// TwinCAT 3 PLC project Untitled1
// ProgramVersion: 3.1.4026.24
// libraries:
//   RobustSolution, * (BATW)
//   Tc2_MC2, * (Beckhoff Automation GmbH)
//   Tc2_Standard, * (Beckhoff Automation GmbH)
//   Tc2_System, * (Beckhoff Automation GmbH)
//   TcUnit, * (www.tcunit.org)
// project tree:
//   GVLs/ GVL_IO.TcGVL (not stored), GVL_Module.TcGVL
//   / PlcTask.TcTTO, UnitTestTask.TcTTO
//   POUs/10_Chamber1/DUTs/Ctrl Status Interface/ ST_Chamber1_CtrlStatus.TcDUT, ST_Chamber1_ServiceCtrl.TcDUT, ST_Chamber1_ServiceParam.TcDUT, ST_Chamber1_ServiceStatus.TcDUT
//   POUs/10_Chamber1/DUTs/ E_Chamber1ErrorCode.TcDUT, E_Chamber1ServiceId.TcDUT
//   POUs/10_Chamber1/DUTs/External IO/ ST_Chamber1_Signal_In.TcDUT (not stored), ST_Chamber1_Signal_Out.TcDUT
//   POUs/10_Chamber1/DUTs/Service Param/PreparePositionService/ E_Chamber1PreparePositionStep.TcDUT (not stored), ST_Chamber1PreparePositionParam.TcDUT
//   POUs/10_Chamber1/DUTs/Service Param/ ST_Chamber1LiftPinAxisMoveAbsParam.TcDUT, ST_Chamber1LiftPinAxisMoveVelParam.TcDUT, ST_Chamber1SpinAxisJogParam.TcDUT, ST_Chamber1SpinAxisMoveAbsParam.TcDUT (not stored), ST_Chamber1SpinAxisMoveVelParam.TcDUT
//   POUs/10_Chamber1/ FB_Chamber1ModuleConfigurationAdapter.TcPOU (not stored), FB_Chamber1_Module.TcPOU
//   POUs/10_Chamber1/Services/ FB_Chamber1LiftPinAxisMoveAbsServices.TcPOU (not stored), FB_Chamber1LiftPinAxisMoveVelCCWServices.TcPOU (not stored), FB_Chamber1LiftPinAxisMoveVelCWServices.TcPOU (not stored), FB_Chamber1PreparePositionService.TcPOU (not stored), FB_Chamber1SpinAxisJogCWServices.TcPOU (not stored), FB_Chamber1SpinAxisMoveAbsServices.TcPOU (not stored), FB_Chamber1SpinAxisMoveVelCWServices.TcPOU (not stored), FB_Chamber1WaferReceiveService.TcPOU (not stored), FB_Chamber1WaferSendService.TcPOU
//   POUs/ FB_ConfigRoot.TcPOU, MAIN.TcPOU
//   Tests/DUTs/ E_FakeAxisOperation.TcDUT (not stored), ST_FakeAxisCall.TcDUT (not stored), ST_FakeAxisScriptStep.TcDUT (not stored)
//   Tests/Fakes/ FB_FakeAxis_BaseUnit.TcPOU (not stored)
//   Tests/ PRG_TEST.TcPOU
//   Tests/Suites/BaseUnit/ FB_FakeAxis_BaseUnitTests.TcPOU (not stored)
//   Tests/Suites/Modules/ FB_Chamber1_ModuleTests.TcPOU
//   Tests/Suites/Services/ FB_Chamber1MoveVelServiceTests.TcPOU, FB_Chamber1SpinAxisMoveAbsServiceTests.TcPOU
// real-time tasks:
//   TASK PlcTask: cycle T#10ms, priority 20, ADS port 350
//   TASK UnitTest Task: cycle T#10ms, priority 1, ADS port 351
// motion (NC):
//   TASK NC-Task 1 SAF: cycle T#2ms, priority 4, ADS port 501
//   TASK NC-Task 1 SVB: cycle T#10ms, priority 8, ADS port 511
//   AXIS Axis 1 (id 1)
//     OtherSettings: AllowMotionCmdToSlave=true
//     encoder EncType=1
//     drive DrvType=5
//       Analog: TorqueSetpointScale=10, ScaleFactorActTorque=0.1
//     controller CtrType=1
//       CtrPara: PriorControlFactor=1
//         Observer: BandWidth=20
//   AXIS Axis 2 (id 2)
//     OtherSettings: AllowMotionCmdToSlave=true
//     encoder EncType=1
//     drive DrvType=5
//       Analog: TorqueSetpointScale=10, ScaleFactorActTorque=0.1
//     controller CtrType=1
//       CtrPara: PriorControlFactor=1
//         Observer: BandWidth=20
// variable links:
//   Untitled1/Untitled1 Instance <-> NC-Task 1 SAF/Axes/Axis 1
//     PlcTask Inputs/GVL_IO.NC_Axis1._Axis.NcToPlc <-> Outputs/ToPlc
//     PlcTask Outputs/GVL_IO.NC_Axis1._Axis.PlcToNc <-> Inputs/FromPlc
//   Untitled1/Untitled1 Instance <-> NC-Task 1 SAF/Axes/Axis 2
//     PlcTask Inputs/GVL_IO.NC_Axis2._Axis.NcToPlc <-> Outputs/ToPlc
//     PlcTask Outputs/GVL_IO.NC_Axis2._Axis.PlcToNc <-> Inputs/FromPlc

CONFIGURATION Untitled1
    RESOURCE PLC ON TwinCAT3
        TASK PlcTask(INTERVAL := T#10ms, PRIORITY := 20);
        TASK UnitTestTask(INTERVAL := T#10ms, PRIORITY := 1);
        PROGRAM MAIN WITH PlcTask : MAIN;
        PROGRAM PRG_TEST WITH UnitTestTask : PRG_TEST;
    END_RESOURCE
END_CONFIGURATION

// ---- POUs/10_Chamber1/DUTs/Ctrl Status Interface/ST_Chamber1_CtrlStatus.TcDUT
TYPE ST_Chamber1_CtrlStatus EXTENDS ST_Module_CtrlStatus_Base :
STRUCT
	ServiceCtrl : ST_Chamber1_ServiceCtrl;
	ServiceParam : ST_Chamber1_ServiceParam;
	ServiceStatus : ST_Chamber1_ServiceStatus;
END_STRUCT
END_TYPE

// ---- POUs/10_Chamber1/DUTs/Ctrl Status Interface/ST_Chamber1_ServiceCtrl.TcDUT
TYPE ST_Chamber1_ServiceCtrl :
STRUCT
	SpinAxisJogCW : ST_ServiceCtrl;
	SpinAxisMoveAbs : ST_ServiceCtrl;
	SpinAxisMoveVelCW	: ST_ServiceCtrl;
	LiftPinAxisMoveVelCW : ST_ServiceCtrl;
	LiftPinAxisMoveVelCCW : ST_ServiceCtrl;
	LiftPinAxisMoveAbs : ST_ServiceCtrl;
	
	WaferSend : ST_ServiceCtrl;
	WaferReceive : ST_ServiceCtrl;
	PreparePosition : ST_ServiceCtrl;
END_STRUCT
END_TYPE

// ---- POUs/10_Chamber1/DUTs/Ctrl Status Interface/ST_Chamber1_ServiceParam.TcDUT
TYPE ST_Chamber1_ServiceParam :
STRUCT
	SpinAxisJogCW : ST_Chamber1SpinAxisJogParam;
	SpinAxisMoveAbs : ST_Chamber1SpinAxisMoveAbsParam;
	SpinAxisMoveVelCW : ST_Chamber1SpinAxisMoveVelParam;
	LiftPinAxisMoveVelCW : ST_Chamber1LiftPinAxisMoveVelParam;
	LiftPinAxisMoveVelCCW : ST_Chamber1LiftPinAxisMoveVelParam;
	LiftPinAxisMoveAbs : ST_Chamber1LiftPinAxisMoveAbsParam;
	WaferReceive : ST_WaferTransferParam;
	WaferSend : ST_WaferTransferParam;
	PreparePosition : ST_Chamber1PreparePositionParam;
END_STRUCT
END_TYPE

// ---- POUs/10_Chamber1/DUTs/Ctrl Status Interface/ST_Chamber1_ServiceStatus.TcDUT
TYPE ST_Chamber1_ServiceStatus :
STRUCT
	SpinAxisJogCW : ST_ServiceStatus;
	SpinAxisMoveAbs : ST_ServiceStatus;
	SpinAxisMoveVelCW : ST_ServiceStatus;
	LiftPinAxisMoveVelCW : ST_ServiceStatus;
	LiftPinAxisMoveVelCCW : ST_ServiceStatus;
	LiftPinAxisMoveAbs : ST_ServiceStatus;
	WaferSend : ST_ServiceStatus;
	WaferReceive : ST_ServiceStatus;
	PreparePosition : ST_ServiceStatus;
END_STRUCT
END_TYPE

// ---- POUs/10_Chamber1/DUTs/E_Chamber1ErrorCode.TcDUT
{attribute 'qualified_only'}
{attribute 'to_string'}
TYPE E_Chamber1ErrorCode :
(
	None := 0,
	Axis_Not_Servo_On_During_Starting := 1,
	Axis_Is_Busy_During_Starting := 2,
	Invalid_Param := 3,
	Axis_Command_Error_During_Execute := 4,
	Error_While_Stop_Axis := 5,
	// The BaseUnit was already owned by another Service.
	Resource_Acquire_Failed_During_Starting := 6,
	// The asynchronous Reset used while aborting failed.
	Error_While_Reset_Axis := 7
)UDINT;
END_TYPE

// ---- POUs/10_Chamber1/DUTs/E_Chamber1ServiceId.TcDUT
{attribute 'qualified_only'}
{attribute 'to_string'}
TYPE E_Chamber1ServiceId :
(
	// Each value identifies one Service instance within the Chamber1 Module.
	None := 0,
	SpinAxisJogCW := 1,
	SpinAxisMoveAbs := 2,
	SpinAxisMoveVelCW := 3,
	LiftPinAxisMoveVelCW := 4,
	LiftPinAxisMoveVelCCW := 5,
	LiftPinAxisMoveAbs := 6,
	WaferSend := 8,
	WaferReceive := 9,
	PreparePosition := 10
) UDINT;
END_TYPE

// ---- POUs/10_Chamber1/DUTs/External IO/ST_Chamber1_Signal_Out.TcDUT
TYPE ST_Chamber1_Signal_Out :
STRUCT
	bVaccumOn : BOOL;

	bDOs : ARRAY[1..16] OF BOOL;
	rAOs : ARRAY[1..16] OF REAL;
END_STRUCT
END_TYPE

// ---- POUs/10_Chamber1/DUTs/Service Param/PreparePositionService/ST_Chamber1PreparePositionParam.TcDUT
TYPE ST_Chamber1PreparePositionParam :
STRUCT
	LiftReady : ST_Chamber1LiftPinAxisMoveAbsParam;
	SpinAlign : ST_Chamber1SpinAxisMoveAbsParam;
	LiftWork : ST_Chamber1LiftPinAxisMoveAbsParam;
END_STRUCT
END_TYPE

// ---- POUs/10_Chamber1/DUTs/Service Param/ST_Chamber1LiftPinAxisMoveAbsParam.TcDUT
TYPE ST_Chamber1LiftPinAxisMoveAbsParam :
STRUCT
	Position : LREAL;
	Velocity : LREAL;
	Acceleration : LREAL;
	Deceleration : LREAL;
END_STRUCT
END_TYPE

// ---- POUs/10_Chamber1/DUTs/Service Param/ST_Chamber1LiftPinAxisMoveVelParam.TcDUT
TYPE ST_Chamber1LiftPinAxisMoveVelParam :
STRUCT
	Velocity : LREAL;
	Acceleration : LREAL;
	Deceleration : LREAL;
END_STRUCT
END_TYPE

// ---- POUs/10_Chamber1/DUTs/Service Param/ST_Chamber1SpinAxisJogParam.TcDUT
TYPE ST_Chamber1SpinAxisJogParam :
STRUCT
	Position : LREAL;
	Velocity : LREAL;
	Acceleration : LREAL;
	Deceleration : LREAL;
END_STRUCT
END_TYPE

// ---- POUs/10_Chamber1/DUTs/Service Param/ST_Chamber1SpinAxisMoveVelParam.TcDUT
TYPE ST_Chamber1SpinAxisMoveVelParam :
STRUCT
	Velocity : LREAL;
	Acceleration : LREAL;
	Deceleration : LREAL;
END_STRUCT
END_TYPE

// ---- GVLs/GVL_Module.TcGVL
{attribute 'qualified_only'}
VAR_GLOBAL
	Chamber1 : ARRAY[1..Param_Config.MaxModulePerType] OF FB_Chamber1_Module;
	Chamber1_Runtime : ARRAY[1..Param_Config.MaxModulePerType] OF ST_ModuleRuntimeConfig;
	Chamber1_Control : ARRAY[1..Param_Config.MaxModulePerType] OF ST_Chamber1_CtrlStatus;
	Chamber1_SpinAxis : ARRAY[1..Param_Config.MaxModulePerType] OF I_Axis_BaseUnit;
	Chamber1_LiftPinAxis : ARRAY[1..Param_Config.MaxModulePerType] OF I_Axis_BaseUnit;
END_VAR

// ---- POUs/MAIN.TcPOU
PROGRAM MAIN
VAR
	ConfigRoot : FB_ConfigRoot;
END_VAR

ConfigRoot.Run();

END_PROGRAM

// ---- POUs/FB_ConfigRoot.TcPOU
FUNCTION_BLOCK FB_ConfigRoot EXTENDS FB_ApplicationConfigRoot
VAR
	_Chamber1ModuleConfigurationAdapter : FB_Chamber1ModuleConfigurationAdapter;
END_VAR

METHOD PROTECTED H_RegisterBaseUnits
M_RegisterBaseUnit(BaseUnit := GVL_IO.NC_Axis1);
M_RegisterBaseUnit(BaseUnit := GVL_IO.NC_Axis2);
END_METHOD

METHOD PROTECTED H_RegisterIo
VAR
	nChannel : DINT;
END_VAR
FOR nChannel := LOWER_BOUND(GVL_IO.Term4_EL1889.Chl, 1)
	TO UPPER_BOUND(GVL_IO.Term4_EL1889.Chl, 1) DO
	IF NOT M_RegisterIoNode(
		Variable := GVL_IO.Term4_EL1889.Chl[nChannel],
		Access := E_VariableAccess.ReadOnly) THEN
		RETURN;
	END_IF
END_FOR

FOR nChannel := LOWER_BOUND(GVL_IO.Term2_EL3602.Chl, 1)
	TO UPPER_BOUND(GVL_IO.Term2_EL3602.Chl, 1) DO
	IF NOT M_RegisterIoNode(
		Variable := GVL_IO.Term2_EL3602.Chl[nChannel],
		Access := E_VariableAccess.ReadOnly) THEN
		RETURN;
	END_IF
END_FOR

FOR nChannel := LOWER_BOUND(GVL_IO.Term3_EL2809.Chl, 1)
	TO UPPER_BOUND(GVL_IO.Term3_EL2809.Chl, 1) DO
	IF NOT M_RegisterIoNode(
		Variable := GVL_IO.Term3_EL2809.Chl[nChannel],
		Access := E_VariableAccess.WriteOnly) THEN
		RETURN;
	END_IF
END_FOR
END_METHOD

METHOD PROTECTED H_RegisterModuleTypes
M_RegisterModuleType(
	ModuleTypeName := 'Chamber1',
	Adapter := _Chamber1ModuleConfigurationAdapter);
END_METHOD

METHOD PROTECTED H_RunModules
VAR_INPUT
	VariableNodeReader : I_VariableNodeReader;
END_VAR
VAR_IN_OUT CONSTANT
	SystemContext : ST_SystemContext;
END_VAR
VAR
	nModule : UINT;
END_VAR
FOR nModule := 1 TO Param_Config.MaxModulePerType DO
	IF GVL_Module.Chamber1_Runtime[nModule].Enabled
		AND GVL_Module.Chamber1_Runtime[nModule].Valid THEN
		GVL_Module.Chamber1[nModule](
			HeartbeatIndex := GVL_Module.Chamber1_Control[nModule].HeartbeatIndex,
			ModuleCtrl := GVL_Module.Chamber1_Control[nModule].ModuleCtrl,
			ServiceCtrl := GVL_Module.Chamber1_Control[nModule].ServiceCtrl,
			ServiceParam := GVL_Module.Chamber1_Control[nModule].ServiceParam,
			SystemContext := SystemContext,
			RuntimeConfig := GVL_Module.Chamber1_Runtime[nModule],
			VariableNodeReader := VariableNodeReader,
			SpinAxis_BaseUnit := GVL_Module.Chamber1_SpinAxis[nModule],
			LiftPinAxis_BaseUnit := GVL_Module.Chamber1_LiftPinAxis[nModule],
			ModuleStatus => GVL_Module.Chamber1_Control[nModule].ModuleStatus,
			ServiceStatus => GVL_Module.Chamber1_Control[nModule].ServiceStatus,
			ModuleAlarmList => GVL_Module.Chamber1_Control[nModule].ModuleAlarmList,
			ModuleDataList => GVL_Module.Chamber1_Control[nModule].ModuleDataList,
			ModuleVariableList => GVL_Module.Chamber1_Control[nModule].ModuleVariableList);
	END_IF
END_FOR
END_METHOD

END_FUNCTION_BLOCK

// ---- Tests/PRG_TEST.TcPOU
PROGRAM PRG_TEST
VAR
	FakeAxisContractTests : FB_FakeAxis_BaseUnitTests;
	
	MoveAbsServiceTests : FB_Chamber1SpinAxisMoveAbsServiceTests;
	MoveVelServiceTests : FB_Chamber1MoveVelServiceTests;
	
	Chamber1ModuleTests : FB_Chamber1_ModuleTests;
END_VAR

TcUnit.RUN();

END_PROGRAM

// ---- Tests/Suites/Services/FB_Chamber1SpinAxisMoveAbsServiceTests.TcPOU
FUNCTION_BLOCK FB_Chamber1SpinAxisMoveAbsServiceTests EXTENDS TcUnit.FB_TestSuite

SuccessfulMoveAbsCompletesAndReleasesAxis();
MoveAbsErrorStopsSafelyAndRecordsError();
InvalidParamStopsStartingWithoutAcquiringAxis();
ResourceAcquireFailureStopsStartingWithoutDisturbingOwner();

METHOD InvalidParamStopsStartingWithoutAcquiringAxis
VAR_INST
	FakeAxis : FB_FakeAxis_BaseUnit;
	Axis : I_Axis_BaseUnit;
	Service : FB_Chamber1SpinAxisMoveAbsServices;
	Ctrl : ST_ServiceCtrl;
	Param : ST_Chamber1SpinAxisMoveAbsParam;
	Context : ST_ServiceContext;
	nPhase : UINT;
END_VAR
TEST('InvalidParamStopsStartingWithoutAcquiringAxis');

CASE nPhase OF
	0:
		// Set invalid param
		FakeAxis.M_ResetScenario();
		Axis := FakeAxis;
		Param.Position := 50;
		Param.Velocity := 0;
		Param.Acceleration := 20;
		Param.Deceleration := 30;
		Context.ModuleId := 1;
		Context.UtcDateTime := '20260813123456007';

		// Cyclic update
		Service(Ctrl := Ctrl, Param := Param, Context := Context, Axis_BaseUnit := Axis, ServiceId := 23);
		FakeAxis.M_CyclicUpdate();

		// Check service run into certain state
		AssertTrue(Condition := Service.PackMLOut.eStateCurrent = E_PackMLState.Aborted, Message := 'Initial scan must reach Aborted.');
		nPhase := 1;

	1:
		// Set PackML cmd: Clear
		Ctrl.PackMLIn.eCommand := E_PackMLCommand.Clear;
		Ctrl.PackMLIn.bCommandChangeRequest := TRUE;

		// Cyclic update
		Service(Ctrl := Ctrl, Param := Param, Context := Context, Axis_BaseUnit := Axis, ServiceId := 23);
		FakeAxis.M_CyclicUpdate();

		// Check service run into certain state
		AssertTrue(Condition := Service.PackMLOut.eStateCurrent = E_PackMLState.Stopped, Message := 'Clear must reach Stopped.');

		// Reset request flag
		Ctrl.PackMLIn.bCommandChangeRequest := FALSE;
		Service(Ctrl := Ctrl, Param := Param, Context := Context, Axis_BaseUnit := Axis, ServiceId := 23);
		FakeAxis.M_CyclicUpdate();

		// Set PackML cmd: Reset
		Ctrl.PackMLIn.eCommand := E_PackMLCommand.Reset;
		Ctrl.PackMLIn.bCommandChangeRequest := TRUE;

		// Cyclic update
		Service(Ctrl := Ctrl, Param := Param, Context := Context, Axis_BaseUnit := Axis, ServiceId := 23);
		FakeAxis.M_CyclicUpdate();

		// Check service run into certain state
		AssertTrue(Condition := Service.PackMLOut.eStateCurrent = E_PackMLState.Idle, Message := 'Reset must reach Idle.');
		nPhase := 2;

	2:
		// Reset request flag
		Ctrl.PackMLIn.bCommandChangeRequest := FALSE;
		Service(Ctrl := Ctrl, Param := Param, Context := Context, Axis_BaseUnit := Axis, ServiceId := 23);
		FakeAxis.M_CyclicUpdate();

		// Set PackML cmd: Start
		Ctrl.PackMLIn.eCommand := E_PackMLCommand.Start;
		Ctrl.PackMLIn.bCommandChangeRequest := TRUE;

		// Cyclic update
		Service(Ctrl := Ctrl, Param := Param, Context := Context, Axis_BaseUnit := Axis, ServiceId := 23);
		FakeAxis.M_CyclicUpdate();

		// Check service remains in Starting until queued Stop is processed
		AssertTrue(Condition := Service.PackMLOut.eStateCurrent = E_PackMLState.Starting, Message := 'Invalid Param must remain in Starting until queued Stop is processed.');

		// Check certain alarm emerged
		AssertTrue(Condition := Service.Status.ErrorList[1].MainErrorId = E_Chamber1ErrorCode.Invalid_Param, Message := 'Invalid Velocity must record Invalid_Param.');
		AssertTrue(Condition := Service.Status.ErrorList[1].SourceErrorId = 0, Message := 'Invalid Param must use SourceErrorId zero.');
		AssertTrue(Condition := Service.Status.ErrorList[1].Message = 'Velocity must be greater than zero.', Message := 'Invalid Velocity must have a specific message.');

		// Check service did not acquire or call the Axis
		AssertFalse(Condition := Axis.M_IsResourceOwner(OwnerId := 23), Message := 'Invalid Param must not acquire Axis ownership.');
		AssertTrue(Condition := FakeAxis.HistoryCount = 0, Message := 'Invalid Param must not issue an Axis command.');
		nPhase := 3;

	3:
		// Reset request flag & process queued Stop
		Ctrl.PackMLIn.bCommandChangeRequest := FALSE;
		Service(Ctrl := Ctrl, Param := Param, Context := Context, Axis_BaseUnit := Axis, ServiceId := 23);
		FakeAxis.M_CyclicUpdate();

		// Check service safely returns to Stopped
		AssertTrue(Condition := Service.PackMLOut.eStateCurrent = E_PackMLState.Stopped, Message := 'Queued Stop must return invalid Starting to Stopped.');

		// Check no duplicate alarm or Axis side effect emerged
		AssertTrue(Condition := Service.Status.ErrorList[1].MainErrorId = E_Chamber1ErrorCode.Invalid_Param, Message := 'Invalid Param must remain recorded after stopping.');
		AssertTrue(Condition := Service.Status.ErrorList[2].MainErrorId = 0, Message := 'Invalid Param must only be recorded once.');
		AssertFalse(Condition := Axis.M_IsResourceOwner(OwnerId := 23), Message := 'Stopped Service must not own the Axis.');
		AssertTrue(Condition := FakeAxis.HistoryCount = 0, Message := 'Stopping without ownership must not issue an Axis command.');
		nPhase := 0;

		TEST_FINISHED();
END_CASE
END_METHOD

METHOD MoveAbsErrorStopsSafelyAndRecordsError
VAR_INST
	FakeAxis : FB_FakeAxis_BaseUnit;
	Axis : I_Axis_BaseUnit;
	Service : FB_Chamber1SpinAxisMoveAbsServices;
	Ctrl : ST_ServiceCtrl;
	Param : ST_Chamber1SpinAxisMoveAbsParam;
	Context : ST_ServiceContext;
	MoveWithdrawalCall : ST_FakeAxisCall;
	StopCall : ST_FakeAxisCall;
	nHistoryBeforeStopping : UINT;
	nPhase : UINT;
END_VAR
TEST('MoveAbsErrorStopsSafelyAndRecordsError');

CASE nPhase OF
	0:
		// Set param
		FakeAxis.M_ResetScenario();
		Axis := FakeAxis;
		Param.Position := 50;
		Param.Velocity := 10;
		Param.Acceleration := 20;
		Param.Deceleration := 30;
		Context.ModuleId := 1;
		Context.UtcDateTime := '20260813123456007';
		
		// Set script: move abs. failed and then stop success
		AssertTrue(
			Condition := FakeAxis.M_QueueResult(
				Operation := E_FakeAxisOperation.MoveAbs,
				AfterActiveCycles := 1,
				Done := FALSE,
				InVelocity := FALSE,
				Error := TRUE,
				ErrorId := 16#1234),
			Message := 'MoveAbs Error script must be accepted.');
		AssertTrue(
			Condition := FakeAxis.M_QueueResult(
				Operation := E_FakeAxisOperation.Stop,
				AfterActiveCycles := 2,
				Done := TRUE,
				InVelocity := FALSE,
				Error := FALSE,
				ErrorId := 0),
			Message := 'Stop Done script must be accepted.');
		
		// Cyclic update
		Service(Ctrl := Ctrl, Param := Param, Context := Context, Axis_BaseUnit := Axis, ServiceId := 22);
		FakeAxis.M_CyclicUpdate();
		nPhase := 1;

	1:
		// Set PackML cmd: Clear
		Ctrl.PackMLIn.eCommand := E_PackMLCommand.Clear;
		Ctrl.PackMLIn.bCommandChangeRequest := TRUE;
		Service(Ctrl := Ctrl, Param := Param, Context := Context, Axis_BaseUnit := Axis, ServiceId := 22);
		FakeAxis.M_CyclicUpdate();

		// Reset request flag
		Ctrl.PackMLIn.bCommandChangeRequest := FALSE;
		Service(Ctrl := Ctrl, Param := Param, Context := Context, Axis_BaseUnit := Axis, ServiceId := 22);
		FakeAxis.M_CyclicUpdate();

		// Set PackML cmd: Reset
		Ctrl.PackMLIn.eCommand := E_PackMLCommand.Reset;
		Ctrl.PackMLIn.bCommandChangeRequest := TRUE;
		Service(Ctrl := Ctrl, Param := Param, Context := Context, Axis_BaseUnit := Axis, ServiceId := 22);
		FakeAxis.M_CyclicUpdate();
		nPhase := 2;

	2:
		// Reset request flag
		Ctrl.PackMLIn.bCommandChangeRequest := FALSE;
		Service(Ctrl := Ctrl, Param := Param, Context := Context, Axis_BaseUnit := Axis, ServiceId := 22);
		FakeAxis.M_CyclicUpdate();

		// Set PackML cmd: Start
		Ctrl.PackMLIn.eCommand := E_PackMLCommand.Start;
		Ctrl.PackMLIn.bCommandChangeRequest := TRUE;
		Service(Ctrl := Ctrl, Param := Param, Context := Context, Axis_BaseUnit := Axis, ServiceId := 22);
		FakeAxis.M_CyclicUpdate();
		AssertTrue(Condition := Service.PackMLOut.eStateCurrent = E_PackMLState.Execute, Message := 'Start must reach Execute.');
		nPhase := 3;

	3:
		// Reset request flag & 1st call of move abs. !!!
		Ctrl.PackMLIn.bCommandChangeRequest := FALSE;
		Service(Ctrl := Ctrl, Param := Param, Context := Context, Axis_BaseUnit := Axis, ServiceId := 22);
		FakeAxis.M_CyclicUpdate();
		AssertTrue(Condition := Service.PackMLOut.eStateCurrent = E_PackMLState.Execute, Message := 'MoveAbs Error is reported after the scripted active scan.');
		nPhase := 4;

	4:
		// 2nd call of move abs., error should happened
		Service(Ctrl := Ctrl, Param := Param, Context := Context, Axis_BaseUnit := Axis, ServiceId := 22);
		FakeAxis.M_CyclicUpdate();
		
		// Check service run into certain state
		AssertTrue(Condition := Service.PackMLOut.eStateCurrent = E_PackMLState.Execute, Message := 'MoveAbs Error must queue Stop for the next scan.');
		
		// Check certain alarm emerged
		AssertTrue(Condition := Service.Status.ErrorList[1].MainErrorId = E_Chamber1ErrorCode.Axis_Command_Error_During_Execute, Message := 'MoveAbs Error must be recorded.');
		AssertTrue(Condition := Service.Status.ErrorList[1].SourceErrorId = 16#1234, Message := 'MoveAbs Error must preserve the Axis source error ID.');
		AssertTrue(Condition := Service.Status.ErrorList[2].MainErrorId = 0, Message := 'MoveAbs Error must only be recorded once.');
		AssertTrue(Condition := Axis.M_IsResourceOwner(OwnerId := 22), Message := 'Queued Stop must retain ownership.');
		nPhase := 5;

	5:
		nHistoryBeforeStopping := FakeAxis.HistoryCount;
		
		// Cyclic update
		Service(Ctrl := Ctrl, Param := Param, Context := Context, Axis_BaseUnit := Axis, ServiceId := 22);
		FakeAxis.M_CyclicUpdate();
		
		// Check service run into certain state
		AssertTrue(Condition := Service.PackMLOut.eStateCurrent = E_PackMLState.Stopping, Message := 'Queued Stop must enter Stopping on the next scan.');
		
		// Check withdrawal move abs. cmd
		AssertTrue(Condition := FakeAxis.M_GetCall(Index := nHistoryBeforeStopping + 1, CallRecord => MoveWithdrawalCall), Message := 'Stopping must record MoveAbs withdrawal.');
		AssertTrue(Condition := MoveWithdrawalCall.Operation = E_FakeAxisOperation.MoveAbs, Message := 'Stopping must withdraw MoveAbs before Stop.');
		AssertTrue(Condition := MoveWithdrawalCall.Accepted, Message := 'MoveAbs withdrawal must be accepted.');
		AssertFalse(Condition := MoveWithdrawalCall.Execute, Message := 'Stopping must set MoveAbs Execute to FALSE.');
		
		// Check stop cmd has been called
		AssertTrue(Condition := FakeAxis.M_GetCall(Index := nHistoryBeforeStopping + 2, CallRecord => StopCall), Message := 'Stopping must record Stop after MoveAbs withdrawal.');
		AssertTrue(Condition := StopCall.Operation = E_FakeAxisOperation.Stop, Message := 'Stopping must issue Stop after MoveAbs withdrawal.');
		AssertTrue(Condition := StopCall.Accepted, Message := 'Stop must be accepted by the owned Axis.');
		AssertTrue(Condition := StopCall.Execute, Message := 'Stop Execute must be TRUE while pending.');
		AssertTrue(Condition := StopCall.Deceleration = Param.Deceleration, Message := 'Stop must preserve Deceleration.');
		AssertTrue(Condition := Axis.M_IsResourceOwner(OwnerId := 22), Message := 'Pending Stop must retain ownership.');
		nPhase := 6;

	6:
		// Cyclic update
		Service(Ctrl := Ctrl, Param := Param, Context := Context, Axis_BaseUnit := Axis, ServiceId := 22);
		FakeAxis.M_CyclicUpdate();
		
		// Stop cmd not finished yet according to script
		AssertTrue(Condition := Service.PackMLOut.eStateCurrent = E_PackMLState.Stopping, Message := 'Stop must remain Stopping until Done feedback is observed.');
		AssertTrue(Condition := Axis.M_IsResourceOwner(OwnerId := 22), Message := 'Stop pending scan must retain ownership.');
		nPhase := 7;

	7:
		// Cyclic update
		Service(Ctrl := Ctrl, Param := Param, Context := Context, Axis_BaseUnit := Axis, ServiceId := 22);
		FakeAxis.M_CyclicUpdate();
		
		// Check service run into certain state
		AssertTrue(Condition := Service.PackMLOut.eStateCurrent = E_PackMLState.Stopped, Message := 'Stop Done must reach Stopped.');
		
		// Check resource has been released
		AssertFalse(Condition := Axis.M_IsResourceOwner(OwnerId := 22), Message := 'Stop Done must release Axis ownership.');
		
		// Check alarm still exist
		AssertTrue(Condition := Service.Status.ErrorList[1].MainErrorId = E_Chamber1ErrorCode.Axis_Command_Error_During_Execute, Message := 'MoveAbs Error must remain recorded after stopping.');
		AssertTrue(Condition := Service.Status.ErrorList[1].SourceErrorId = 16#1234, Message := 'Recorded MoveAbs source error ID must remain unchanged.');
		AssertTrue(Condition := Service.Status.ErrorList[2].MainErrorId = 0, Message := 'Repeated scans must not duplicate the MoveAbs Error.');
		
		// Check withdrawal stop cmd
		AssertTrue(Condition := FakeAxis.M_GetCall(Index := FakeAxis.HistoryCount, CallRecord => StopCall), Message := 'Stop falling edge must be recorded.');
		AssertTrue(Condition := StopCall.Operation = E_FakeAxisOperation.Stop, Message := 'Final cleanup call must be Stop.');
		AssertTrue(Condition := StopCall.Accepted, Message := 'Stop falling edge must occur before ownership is released.');
		AssertFalse(Condition := StopCall.Execute, Message := 'Stop Done must set Stop Execute to FALSE.');
		AssertFalse(Condition := FakeAxis.HistoryOverflowed, Message := 'Fake Axis call history must not overflow.');
		nPhase := 0;
		
		TEST_FINISHED();
END_CASE
END_METHOD

METHOD ResourceAcquireFailureStopsStartingWithoutDisturbingOwner
VAR_INST
	FakeAxis : FB_FakeAxis_BaseUnit;
	Axis : I_Axis_BaseUnit;
	Service : FB_Chamber1SpinAxisMoveAbsServices;
	Ctrl : ST_ServiceCtrl;
	Param : ST_Chamber1SpinAxisMoveAbsParam;
	Context : ST_ServiceContext;
	nPhase : UINT;
END_VAR
TEST('ResourceAcquireFailureStopsStartingWithoutDisturbingOwner');

CASE nPhase OF
	0:
		// Set valid param
		FakeAxis.M_ResetScenario();
		Axis := FakeAxis;
		Param.Position := 50;
		Param.Velocity := 10;
		Param.Acceleration := 20;
		Param.Deceleration := 30;
		Context.ModuleId := 1;
		Context.UtcDateTime := '20260813123456007';

		// Cyclic update
		Service(Ctrl := Ctrl, Param := Param, Context := Context, Axis_BaseUnit := Axis, ServiceId := 24);
		FakeAxis.M_CyclicUpdate();

		// Check service run into certain state
		AssertTrue(Condition := Service.PackMLOut.eStateCurrent = E_PackMLState.Aborted, Message := 'Initial scan must reach Aborted.');
		nPhase := 1;

	1:
		// Set PackML cmd: Clear
		Ctrl.PackMLIn.eCommand := E_PackMLCommand.Clear;
		Ctrl.PackMLIn.bCommandChangeRequest := TRUE;

		// Cyclic update
		Service(Ctrl := Ctrl, Param := Param, Context := Context, Axis_BaseUnit := Axis, ServiceId := 24);
		FakeAxis.M_CyclicUpdate();

		// Check service run into certain state
		AssertTrue(Condition := Service.PackMLOut.eStateCurrent = E_PackMLState.Stopped, Message := 'Clear must reach Stopped.');

		// Reset request flag
		Ctrl.PackMLIn.bCommandChangeRequest := FALSE;
		Service(Ctrl := Ctrl, Param := Param, Context := Context, Axis_BaseUnit := Axis, ServiceId := 24);
		FakeAxis.M_CyclicUpdate();

		// Set PackML cmd: Reset
		Ctrl.PackMLIn.eCommand := E_PackMLCommand.Reset;
		Ctrl.PackMLIn.bCommandChangeRequest := TRUE;

		// Cyclic update
		Service(Ctrl := Ctrl, Param := Param, Context := Context, Axis_BaseUnit := Axis, ServiceId := 24);
		FakeAxis.M_CyclicUpdate();

		// Check service run into certain state
		AssertTrue(Condition := Service.PackMLOut.eStateCurrent = E_PackMLState.Idle, Message := 'Reset must reach Idle.');
		nPhase := 2;

	2:
		// Reset request flag
		Ctrl.PackMLIn.bCommandChangeRequest := FALSE;
		Service(Ctrl := Ctrl, Param := Param, Context := Context, Axis_BaseUnit := Axis, ServiceId := 24);
		FakeAxis.M_CyclicUpdate();

		// Reserve the Axis with another owner
		AssertTrue(Condition := Axis.M_AcquireResource(OwnerId := 99), Message := 'Another owner must reserve the Axis.');

		// Set PackML cmd: Start
		Ctrl.PackMLIn.eCommand := E_PackMLCommand.Start;
		Ctrl.PackMLIn.bCommandChangeRequest := TRUE;

		// Cyclic update
		Service(Ctrl := Ctrl, Param := Param, Context := Context, Axis_BaseUnit := Axis, ServiceId := 24);
		FakeAxis.M_CyclicUpdate();

		// Check service remains in Starting until queued Stop is processed
		AssertTrue(Condition := Service.PackMLOut.eStateCurrent = E_PackMLState.Starting, Message := 'Resource acquire failure must remain in Starting until queued Stop is processed.');

		// Check certain alarm emerged
		AssertTrue(Condition := Service.Status.ErrorList[1].MainErrorId = E_Chamber1ErrorCode.Resource_Acquire_Failed_During_Starting, Message := 'Resource contention must be recorded.');
		AssertTrue(Condition := Service.Status.ErrorList[1].SourceErrorId = 0, Message := 'Resource contention must use SourceErrorId zero.');

		// Check existing ownership was not disturbed
		AssertFalse(Condition := Axis.M_IsResourceOwner(OwnerId := 24), Message := 'Service must not acquire the reserved Axis.');
		AssertTrue(Condition := Axis.M_IsResourceOwner(OwnerId := 99), Message := 'Existing Axis owner must remain unchanged.');
		AssertTrue(Condition := FakeAxis.HistoryCount = 0, Message := 'Acquire failure must not issue an Axis command.');
		nPhase := 3;

	3:
		// Reset request flag & process queued Stop
		Ctrl.PackMLIn.bCommandChangeRequest := FALSE;
		Service(Ctrl := Ctrl, Param := Param, Context := Context, Axis_BaseUnit := Axis, ServiceId := 24);
		FakeAxis.M_CyclicUpdate();

		// Check service safely returns to Stopped
		AssertTrue(Condition := Service.PackMLOut.eStateCurrent = E_PackMLState.Stopped, Message := 'Queued Stop must return resource failure to Stopped.');

		// Check existing ownership and alarm remain unchanged
		AssertFalse(Condition := Axis.M_IsResourceOwner(OwnerId := 24), Message := 'Stopped Service must not own the Axis.');
		AssertTrue(Condition := Axis.M_IsResourceOwner(OwnerId := 99), Message := 'Stopping must not release another owner resource.');
		AssertTrue(Condition := Service.Status.ErrorList[1].MainErrorId = E_Chamber1ErrorCode.Resource_Acquire_Failed_During_Starting, Message := 'Resource contention must remain recorded after stopping.');
		AssertTrue(Condition := Service.Status.ErrorList[2].MainErrorId = 0, Message := 'Resource contention must only be recorded once.');
		AssertTrue(Condition := FakeAxis.HistoryCount = 0, Message := 'Stopping without ownership must not issue an Axis command.');
		nPhase := 0;

		TEST_FINISHED();
END_CASE
END_METHOD

METHOD SuccessfulMoveAbsCompletesAndReleasesAxis
VAR_INST
	FakeAxis : FB_FakeAxis_BaseUnit;
	Axis : I_Axis_BaseUnit;
	Service : FB_Chamber1SpinAxisMoveAbsServices;
	Ctrl : ST_ServiceCtrl;
	Param : ST_Chamber1SpinAxisMoveAbsParam;
	Context : ST_ServiceContext;
	CallRecord : ST_FakeAxisCall;
	nPhase : UINT;
END_VAR
TEST('SuccessfulMoveAbsCompletesAndReleasesAxis');

CASE nPhase OF
	0:
		// Set param
		FakeAxis.M_ResetScenario();
		Axis := FakeAxis;
		Param.Position := 125.25;
		Param.Velocity := 15;
		Param.Acceleration := 25;
		Param.Deceleration := 35;
		Context.ModuleId := 1;
		Context.UtcDateTime := '20260813123456007';
		
		// Set script
		AssertTrue(
			Condition := FakeAxis.M_QueueResult(
				Operation := E_FakeAxisOperation.MoveAbs,
				AfterActiveCycles := 2,
				Done := TRUE,
				InVelocity := FALSE,
				Error := FALSE,
				ErrorId := 0),
			Message := 'MoveAbs Done script must be accepted.');
		
		// Cyclic update
		Service(Ctrl := Ctrl, Param := Param, Context := Context, Axis_BaseUnit := Axis, ServiceId := 21);
		FakeAxis.M_CyclicUpdate();
		
		// Check service run into certain state
		AssertTrue(Condition := Service.PackMLOut.eStateCurrent = E_PackMLState.Aborted, Message := 'Initial scan must reach Aborted.');
		nPhase := 1;

	1:
		// Set PackML cmd: Clear
		Ctrl.PackMLIn.eCommand := E_PackMLCommand.Clear;
		Ctrl.PackMLIn.bCommandChangeRequest := TRUE;
		
		// Cyclic update
		Service(Ctrl := Ctrl, Param := Param, Context := Context, Axis_BaseUnit := Axis, ServiceId := 21);
		FakeAxis.M_CyclicUpdate();
		
		// Check service run into certain state
		AssertTrue(Condition := Service.PackMLOut.eStateCurrent = E_PackMLState.Stopped, Message := 'Clear must reach Stopped.');
		
		// Reset request flag
		Ctrl.PackMLIn.bCommandChangeRequest := FALSE;
		Service(Ctrl := Ctrl, Param := Param, Context := Context, Axis_BaseUnit := Axis, ServiceId := 21);
		FakeAxis.M_CyclicUpdate();

		// Set PackML cmd: Reset
		Ctrl.PackMLIn.eCommand := E_PackMLCommand.Reset;
		Ctrl.PackMLIn.bCommandChangeRequest := TRUE;
		
		// Cyclic update
		Service(Ctrl := Ctrl, Param := Param, Context := Context, Axis_BaseUnit := Axis, ServiceId := 21);
		FakeAxis.M_CyclicUpdate();
		
		// Check service run into certain state
		AssertTrue(Condition := Service.PackMLOut.eStateCurrent = E_PackMLState.Idle, Message := 'Reset must reach Idle.');
		nPhase := 2;

	2:
		// Reset request flag
		Ctrl.PackMLIn.bCommandChangeRequest := FALSE;
		Service(Ctrl := Ctrl, Param := Param, Context := Context, Axis_BaseUnit := Axis, ServiceId := 21);
		FakeAxis.M_CyclicUpdate();
		
		// Set PackML cmd: Start
		Ctrl.PackMLIn.eCommand := E_PackMLCommand.Start;
		Ctrl.PackMLIn.bCommandChangeRequest := TRUE;
		
		// Cyclic update
		Service(Ctrl := Ctrl, Param := Param, Context := Context, Axis_BaseUnit := Axis, ServiceId := 21);
		FakeAxis.M_CyclicUpdate();
		
		// Check service run into certain state
		AssertTrue(Condition := Service.PackMLOut.eStateCurrent = E_PackMLState.Execute, Message := 'Start must reach Execute.');
		// Check service get resource
		AssertTrue(Condition := Axis.M_IsResourceOwner(OwnerId := 21), Message := 'Execute must own the Axis.');
		nPhase := 3;

	3:
		// Reset request flag & 1st call of move abs. !!!
		Ctrl.PackMLIn.bCommandChangeRequest := FALSE;
		Service(Ctrl := Ctrl, Param := Param, Context := Context, Axis_BaseUnit := Axis, ServiceId := 21);
		FakeAxis.M_CyclicUpdate();
		
		// Check called cmd is correct
		AssertTrue(Condition := FakeAxis.M_GetCall(Index := FakeAxis.HistoryCount, CallRecord => CallRecord), Message := 'MoveAbs command must be recorded.');
		AssertTrue(Condition := CallRecord.Operation = E_FakeAxisOperation.MoveAbs, Message := 'Execute must issue MoveAbs.');
		AssertTrue(Condition := CallRecord.Accepted, Message := 'MoveAbs must be accepted by the owned Axis.');
		AssertTrue(Condition := CallRecord.Execute, Message := 'MoveAbs Execute must be TRUE.');
		AssertTrue(Condition := CallRecord.OwnerId = 21, Message := 'MoveAbs must use the Service owner ID.');
		AssertTrue(Condition := CallRecord.Position = Param.Position, Message := 'MoveAbs must preserve Position.');
		AssertTrue(Condition := CallRecord.Velocity = Param.Velocity, Message := 'MoveAbs must preserve Velocity.');
		AssertTrue(Condition := CallRecord.Acceleration = Param.Acceleration, Message := 'MoveAbs must preserve Acceleration.');
		AssertTrue(Condition := CallRecord.Deceleration = Param.Deceleration, Message := 'MoveAbs must preserve Deceleration.');
		nPhase := 4;

	4:
		// 2nd call of move abs.
		Service(Ctrl := Ctrl, Param := Param, Context := Context, Axis_BaseUnit := Axis, ServiceId := 21);
		FakeAxis.M_CyclicUpdate();
		AssertTrue(Condition := Service.PackMLOut.eStateCurrent = E_PackMLState.Execute, Message := 'Pending MoveAbs must remain in Execute.');
		AssertTrue(Condition := Axis.M_IsResourceOwner(OwnerId := 21), Message := 'Pending MoveAbs must retain ownership.');
		nPhase := 5;

	5:
		// 3rd call of move abs.
		Service(Ctrl := Ctrl, Param := Param, Context := Context, Axis_BaseUnit := Axis, ServiceId := 21);
		FakeAxis.M_CyclicUpdate();
		
		// Check service run into certain state
		AssertTrue(Condition := Service.PackMLOut.eStateCurrent = E_PackMLState.Completing, Message := 'MoveAbs Done must enter Completing.');
		
		// Check still own the resource
		AssertTrue(Condition := Axis.M_IsResourceOwner(OwnerId := 21), Message := 'Completing entry must retain ownership until MoveAbs is withdrawn.');
		nPhase := 6;

	6:
		// Cyclic update
		Service(Ctrl := Ctrl, Param := Param, Context := Context, Axis_BaseUnit := Axis, ServiceId := 21);
		FakeAxis.M_CyclicUpdate();
		
		// Check service run into certain state
		AssertTrue(Condition := Service.PackMLOut.eStateCurrent = E_PackMLState.Complete, Message := 'Completing must reach Complete.');
		
		// Check release the resource
		AssertFalse(Condition := Axis.M_IsResourceOwner(OwnerId := 21), Message := 'Complete must release Axis ownership.');
		AssertTrue(Condition := Service.Status.ErrorList[1].MainErrorId = 0, Message := 'Successful MoveAbs must not create a Service error.');
		AssertTrue(Condition := FakeAxis.M_GetCall(Index := FakeAxis.HistoryCount, CallRecord => CallRecord), Message := 'MoveAbs withdrawal must be recorded.');
		AssertTrue(Condition := CallRecord.Operation = E_FakeAxisOperation.MoveAbs, Message := 'Completing must withdraw MoveAbs.');
		AssertTrue(Condition := CallRecord.Accepted, Message := 'MoveAbs withdrawal must occur before ownership is released.');
		AssertFalse(Condition := CallRecord.Execute, Message := 'Completing must set MoveAbs Execute to FALSE.');
		AssertFalse(Condition := FakeAxis.HistoryOverflowed, Message := 'Fake Axis call history must not overflow.');
		nPhase := 0;
		
		TEST_FINISHED();
END_CASE
END_METHOD

END_FUNCTION_BLOCK

// ---- Tests/Suites/Services/FB_Chamber1MoveVelServiceTests.TcPOU
FUNCTION_BLOCK FB_Chamber1MoveVelServiceTests EXTENDS TcUnit.FB_TestSuite
VAR
	// Keep large FB instances at Test Suite scope to avoid Method stack overflow.
	SpinService : FB_Chamber1SpinAxisMoveVelCWServices;
	SpinFake : FB_FakeAxis_BaseUnit;
	LiftCWService : FB_Chamber1LiftPinAxisMoveVelCWServices;
	LiftCWFake : FB_FakeAxis_BaseUnit;
	LiftCCWService : FB_Chamber1LiftPinAxisMoveVelCCWServices;
	LiftCCWFake : FB_FakeAxis_BaseUnit;
	ResetService : FB_Chamber1SpinAxisMoveVelCWServices;
	ResetFake : FB_FakeAxis_BaseUnit;
END_VAR

MoveVelServicesCompleteNaturallyWithoutRetrigger();
ResetToIdleKeepsOwnershipUntilStop();

METHOD MoveVelServicesCompleteNaturallyWithoutRetrigger
VAR_INST
	SpinAxis : I_Axis_BaseUnit;
	LiftCWAxis : I_Axis_BaseUnit;
	LiftCCWAxis : I_Axis_BaseUnit;
	Ctrl : ST_ServiceCtrl;
	SpinParam : ST_Chamber1SpinAxisMoveVelParam;
	LiftCWParam : ST_Chamber1LiftPinAxisMoveVelParam;
	LiftCCWParam : ST_Chamber1LiftPinAxisMoveVelParam;
	Context : ST_ServiceContext;
	SpinCall : ST_FakeAxisCall;
	LiftCWCall : ST_FakeAxisCall;
	LiftCCWCall : ST_FakeAxisCall;
	nSpinHistoryBeforeStop : UINT;
	nLiftCWHistoryBeforeStop : UINT;
	nLiftCCWHistoryBeforeStop : UINT;
	nPhase : UINT;
END_VAR
TEST('MoveVelServicesCompleteNaturallyWithoutRetrigger');

CASE nPhase OF
	0:
		SpinFake.M_ResetScenario();
		LiftCWFake.M_ResetScenario();
		LiftCCWFake.M_ResetScenario();
		SpinAxis := SpinFake;
		LiftCWAxis := LiftCWFake;
		LiftCCWAxis := LiftCCWFake;

		SpinParam.Velocity := 11;
		SpinParam.Acceleration := 12;
		SpinParam.Deceleration := 13;
		LiftCWParam.Velocity := 21;
		LiftCWParam.Acceleration := 22;
		LiftCWParam.Deceleration := 23;
		LiftCCWParam.Velocity := 31;
		LiftCCWParam.Acceleration := 32;
		LiftCCWParam.Deceleration := 33;
		Context.ModuleId := 1;

		AssertTrue(Condition := SpinFake.M_QueueResult(Operation := E_FakeAxisOperation.MoveVel, AfterActiveCycles := 2, Done := FALSE, InVelocity := TRUE, Error := FALSE, ErrorId := 0), Message := 'Spin MoveVel script must be accepted.');
		AssertTrue(Condition := LiftCWFake.M_QueueResult(Operation := E_FakeAxisOperation.MoveVel, AfterActiveCycles := 2, Done := FALSE, InVelocity := TRUE, Error := FALSE, ErrorId := 0), Message := 'Lift CW MoveVel script must be accepted.');
		AssertTrue(Condition := LiftCCWFake.M_QueueResult(Operation := E_FakeAxisOperation.MoveVel, AfterActiveCycles := 2, Done := FALSE, InVelocity := TRUE, Error := FALSE, ErrorId := 0), Message := 'Lift CCW MoveVel script must be accepted.');
		AssertTrue(Condition := SpinFake.M_QueueResult(Operation := E_FakeAxisOperation.Stop, AfterActiveCycles := 1, Done := TRUE, InVelocity := FALSE, Error := FALSE, ErrorId := 0), Message := 'Spin Stop script must be accepted.');
		AssertTrue(Condition := LiftCWFake.M_QueueResult(Operation := E_FakeAxisOperation.Stop, AfterActiveCycles := 1, Done := TRUE, InVelocity := FALSE, Error := FALSE, ErrorId := 0), Message := 'Lift CW Stop script must be accepted.');
		AssertTrue(Condition := LiftCCWFake.M_QueueResult(Operation := E_FakeAxisOperation.Stop, AfterActiveCycles := 1, Done := TRUE, InVelocity := FALSE, Error := FALSE, ErrorId := 0), Message := 'Lift CCW Stop script must be accepted.');

		SpinService(Ctrl := Ctrl, Param := SpinParam, Context := Context, Axis_BaseUnit := SpinAxis, ServiceId := 31);
		LiftCWService(Ctrl := Ctrl, Param := LiftCWParam, Context := Context, Axis_BaseUnit := LiftCWAxis, ServiceId := 32);
		LiftCCWService(Ctrl := Ctrl, Param := LiftCCWParam, Context := Context, Axis_BaseUnit := LiftCCWAxis, ServiceId := 33);
		SpinFake.M_CyclicUpdate();
		LiftCWFake.M_CyclicUpdate();
		LiftCCWFake.M_CyclicUpdate();

		AssertTrue(Condition := (SpinService.PackMLOut.eStateCurrent = E_PackMLState.Aborted)
			AND (LiftCWService.PackMLOut.eStateCurrent = E_PackMLState.Aborted)
			AND (LiftCCWService.PackMLOut.eStateCurrent = E_PackMLState.Aborted), Message := 'Initial scan must reach Aborted.');
		AssertTrue(Condition := (SpinService.Status.CompletionBehavior = E_ServiceCompletionBehavior.NaturalCompletion)
			AND (LiftCWService.Status.CompletionBehavior = E_ServiceCompletionBehavior.NaturalCompletion)
			AND (LiftCCWService.Status.CompletionBehavior = E_ServiceCompletionBehavior.NaturalCompletion), Message := 'Every MoveVel Service must publish NaturalCompletion.');
		nPhase := 1;

	1:
		Ctrl.PackMLIn.eCommand := E_PackMLCommand.Clear;
		Ctrl.PackMLIn.bCommandChangeRequest := TRUE;
		SpinService(Ctrl := Ctrl, Param := SpinParam, Context := Context, Axis_BaseUnit := SpinAxis, ServiceId := 31);
		LiftCWService(Ctrl := Ctrl, Param := LiftCWParam, Context := Context, Axis_BaseUnit := LiftCWAxis, ServiceId := 32);
		LiftCCWService(Ctrl := Ctrl, Param := LiftCCWParam, Context := Context, Axis_BaseUnit := LiftCCWAxis, ServiceId := 33);
		SpinFake.M_CyclicUpdate();
		LiftCWFake.M_CyclicUpdate();
		LiftCCWFake.M_CyclicUpdate();
		AssertTrue(Condition := (SpinService.PackMLOut.eStateCurrent = E_PackMLState.Stopped)
			AND (LiftCWService.PackMLOut.eStateCurrent = E_PackMLState.Stopped)
			AND (LiftCCWService.PackMLOut.eStateCurrent = E_PackMLState.Stopped), Message := 'Clear must bring every MoveVel Service to Stopped.');

		Ctrl.PackMLIn.bCommandChangeRequest := FALSE;
		SpinService(Ctrl := Ctrl, Param := SpinParam, Context := Context, Axis_BaseUnit := SpinAxis, ServiceId := 31);
		LiftCWService(Ctrl := Ctrl, Param := LiftCWParam, Context := Context, Axis_BaseUnit := LiftCWAxis, ServiceId := 32);
		LiftCCWService(Ctrl := Ctrl, Param := LiftCCWParam, Context := Context, Axis_BaseUnit := LiftCCWAxis, ServiceId := 33);
		SpinFake.M_CyclicUpdate();
		LiftCWFake.M_CyclicUpdate();
		LiftCCWFake.M_CyclicUpdate();

		Ctrl.PackMLIn.eCommand := E_PackMLCommand.Reset;
		Ctrl.PackMLIn.bCommandChangeRequest := TRUE;
		SpinService(Ctrl := Ctrl, Param := SpinParam, Context := Context, Axis_BaseUnit := SpinAxis, ServiceId := 31);
		LiftCWService(Ctrl := Ctrl, Param := LiftCWParam, Context := Context, Axis_BaseUnit := LiftCWAxis, ServiceId := 32);
		LiftCCWService(Ctrl := Ctrl, Param := LiftCCWParam, Context := Context, Axis_BaseUnit := LiftCCWAxis, ServiceId := 33);
		SpinFake.M_CyclicUpdate();
		LiftCWFake.M_CyclicUpdate();
		LiftCCWFake.M_CyclicUpdate();
		AssertTrue(Condition := (SpinService.PackMLOut.eStateCurrent = E_PackMLState.Idle)
			AND (LiftCWService.PackMLOut.eStateCurrent = E_PackMLState.Idle)
			AND (LiftCCWService.PackMLOut.eStateCurrent = E_PackMLState.Idle), Message := 'Reset must bring every MoveVel Service to Idle.');
		nPhase := 2;

	2:
		Ctrl.PackMLIn.bCommandChangeRequest := FALSE;
		SpinService(Ctrl := Ctrl, Param := SpinParam, Context := Context, Axis_BaseUnit := SpinAxis, ServiceId := 31);
		LiftCWService(Ctrl := Ctrl, Param := LiftCWParam, Context := Context, Axis_BaseUnit := LiftCWAxis, ServiceId := 32);
		LiftCCWService(Ctrl := Ctrl, Param := LiftCCWParam, Context := Context, Axis_BaseUnit := LiftCCWAxis, ServiceId := 33);
		SpinFake.M_CyclicUpdate();
		LiftCWFake.M_CyclicUpdate();
		LiftCCWFake.M_CyclicUpdate();

		Ctrl.PackMLIn.eCommand := E_PackMLCommand.Start;
		Ctrl.PackMLIn.bCommandChangeRequest := TRUE;
		SpinService(Ctrl := Ctrl, Param := SpinParam, Context := Context, Axis_BaseUnit := SpinAxis, ServiceId := 31);
		LiftCWService(Ctrl := Ctrl, Param := LiftCWParam, Context := Context, Axis_BaseUnit := LiftCWAxis, ServiceId := 32);
		LiftCCWService(Ctrl := Ctrl, Param := LiftCCWParam, Context := Context, Axis_BaseUnit := LiftCCWAxis, ServiceId := 33);
		SpinFake.M_CyclicUpdate();
		LiftCWFake.M_CyclicUpdate();
		LiftCCWFake.M_CyclicUpdate();
		AssertTrue(Condition := (SpinService.PackMLOut.eStateCurrent = E_PackMLState.Execute)
			AND (LiftCWService.PackMLOut.eStateCurrent = E_PackMLState.Execute)
			AND (LiftCCWService.PackMLOut.eStateCurrent = E_PackMLState.Execute), Message := 'Valid Start must bring every MoveVel Service to Execute.');
		AssertTrue(Condition := SpinAxis.M_IsResourceOwner(OwnerId := 31)
			AND LiftCWAxis.M_IsResourceOwner(OwnerId := 32)
			AND LiftCCWAxis.M_IsResourceOwner(OwnerId := 33), Message := 'Execute must retain each Axis ownership.');
		nPhase := 3;

	3:
		Ctrl.PackMLIn.bCommandChangeRequest := FALSE;
		SpinService(Ctrl := Ctrl, Param := SpinParam, Context := Context, Axis_BaseUnit := SpinAxis, ServiceId := 31);
		LiftCWService(Ctrl := Ctrl, Param := LiftCWParam, Context := Context, Axis_BaseUnit := LiftCWAxis, ServiceId := 32);
		LiftCCWService(Ctrl := Ctrl, Param := LiftCCWParam, Context := Context, Axis_BaseUnit := LiftCCWAxis, ServiceId := 33);
		SpinFake.M_CyclicUpdate();
		LiftCWFake.M_CyclicUpdate();
		LiftCCWFake.M_CyclicUpdate();

		AssertTrue(Condition := SpinFake.M_GetCall(Index := SpinFake.HistoryCount, CallRecord => SpinCall), Message := 'Spin MoveVel call must be recorded.');
		AssertTrue(Condition := LiftCWFake.M_GetCall(Index := LiftCWFake.HistoryCount, CallRecord => LiftCWCall), Message := 'Lift CW MoveVel call must be recorded.');
		AssertTrue(Condition := LiftCCWFake.M_GetCall(Index := LiftCCWFake.HistoryCount, CallRecord => LiftCCWCall), Message := 'Lift CCW MoveVel call must be recorded.');
		AssertTrue(Condition := SpinCall.Execute AND LiftCWCall.Execute AND LiftCCWCall.Execute, Message := 'Initial MoveVel requests must remain high.');
		AssertTrue(Condition := (SpinCall.Direction = MC_Direction.MC_Positive_Direction)
			AND (LiftCWCall.Direction = MC_Direction.MC_Positive_Direction)
			AND (LiftCCWCall.Direction = MC_Direction.MC_Negative_Direction), Message := 'MoveVel Services must preserve their configured directions.');

		// Mutations after Start must not change the active command snapshot.
		SpinParam.Velocity := 111;
		SpinParam.Acceleration := 112;
		SpinParam.Deceleration := 113;
		LiftCWParam.Velocity := 121;
		LiftCWParam.Acceleration := 122;
		LiftCWParam.Deceleration := 123;
		LiftCCWParam.Velocity := 131;
		LiftCCWParam.Acceleration := 132;
		LiftCCWParam.Deceleration := 133;
		nPhase := 4;

	4:
		SpinService(Ctrl := Ctrl, Param := SpinParam, Context := Context, Axis_BaseUnit := SpinAxis, ServiceId := 31);
		LiftCWService(Ctrl := Ctrl, Param := LiftCWParam, Context := Context, Axis_BaseUnit := LiftCWAxis, ServiceId := 32);
		LiftCCWService(Ctrl := Ctrl, Param := LiftCCWParam, Context := Context, Axis_BaseUnit := LiftCCWAxis, ServiceId := 33);
		SpinFake.M_CyclicUpdate();
		LiftCWFake.M_CyclicUpdate();
		LiftCCWFake.M_CyclicUpdate();

		AssertTrue(Condition := (SpinService.PackMLOut.eStateCurrent = E_PackMLState.Execute)
			AND (LiftCWService.PackMLOut.eStateCurrent = E_PackMLState.Execute)
			AND (LiftCCWService.PackMLOut.eStateCurrent = E_PackMLState.Execute), Message := 'MoveVel Services must wait for InVelocity.');
		AssertTrue(Condition := SpinFake.M_GetCall(Index := SpinFake.HistoryCount, CallRecord => SpinCall), Message := 'Second Spin MoveVel call must be recorded.');
		AssertTrue(Condition := LiftCWFake.M_GetCall(Index := LiftCWFake.HistoryCount, CallRecord => LiftCWCall), Message := 'Second Lift CW MoveVel call must be recorded.');
		AssertTrue(Condition := LiftCCWFake.M_GetCall(Index := LiftCCWFake.HistoryCount, CallRecord => LiftCCWCall), Message := 'Second Lift CCW MoveVel call must be recorded.');
		AssertTrue(Condition := SpinCall.Execute AND (SpinCall.Velocity = 11) AND (SpinCall.Acceleration = 12) AND (SpinCall.Deceleration = 13), Message := 'Spin MoveVel must keep its Start-time parameters without retriggering.');
		AssertTrue(Condition := LiftCWCall.Execute AND (LiftCWCall.Velocity = 21) AND (LiftCWCall.Acceleration = 22) AND (LiftCWCall.Deceleration = 23), Message := 'Lift CW MoveVel must keep its Start-time parameters without retriggering.');
		AssertTrue(Condition := LiftCCWCall.Execute AND (LiftCCWCall.Velocity = 31) AND (LiftCCWCall.Acceleration = 32) AND (LiftCCWCall.Deceleration = 33), Message := 'Lift CCW MoveVel must keep its Start-time parameters without retriggering.');
		nPhase := 5;

	5:
		SpinService(Ctrl := Ctrl, Param := SpinParam, Context := Context, Axis_BaseUnit := SpinAxis, ServiceId := 31);
		LiftCWService(Ctrl := Ctrl, Param := LiftCWParam, Context := Context, Axis_BaseUnit := LiftCWAxis, ServiceId := 32);
		LiftCCWService(Ctrl := Ctrl, Param := LiftCCWParam, Context := Context, Axis_BaseUnit := LiftCCWAxis, ServiceId := 33);
		SpinFake.M_CyclicUpdate();
		LiftCWFake.M_CyclicUpdate();
		LiftCCWFake.M_CyclicUpdate();
		AssertTrue(Condition := (SpinService.PackMLOut.eStateCurrent = E_PackMLState.Completing)
			AND (LiftCWService.PackMLOut.eStateCurrent = E_PackMLState.Completing)
			AND (LiftCCWService.PackMLOut.eStateCurrent = E_PackMLState.Completing), Message := 'InVelocity must move every MoveVel Service to Completing.');
		AssertTrue(Condition := SpinAxis.M_IsResourceOwner(OwnerId := 31)
			AND LiftCWAxis.M_IsResourceOwner(OwnerId := 32)
			AND LiftCCWAxis.M_IsResourceOwner(OwnerId := 33), Message := 'Completing entry must retain ownership until MoveVel withdrawal.');
		nPhase := 6;

	6:
		SpinService(Ctrl := Ctrl, Param := SpinParam, Context := Context, Axis_BaseUnit := SpinAxis, ServiceId := 31);
		LiftCWService(Ctrl := Ctrl, Param := LiftCWParam, Context := Context, Axis_BaseUnit := LiftCWAxis, ServiceId := 32);
		LiftCCWService(Ctrl := Ctrl, Param := LiftCCWParam, Context := Context, Axis_BaseUnit := LiftCCWAxis, ServiceId := 33);
		SpinFake.M_CyclicUpdate();
		LiftCWFake.M_CyclicUpdate();
		LiftCCWFake.M_CyclicUpdate();

		AssertTrue(Condition := (SpinService.PackMLOut.eStateCurrent = E_PackMLState.Complete)
			AND (LiftCWService.PackMLOut.eStateCurrent = E_PackMLState.Complete)
			AND (LiftCCWService.PackMLOut.eStateCurrent = E_PackMLState.Complete), Message := 'Completing must reach Complete.');
		AssertTrue(Condition := SpinAxis.M_IsResourceOwner(OwnerId := 31)
			AND LiftCWAxis.M_IsResourceOwner(OwnerId := 32)
			AND LiftCCWAxis.M_IsResourceOwner(OwnerId := 33), Message := 'Complete must retain Axis ownership while physical motion continues.');
		AssertTrue(Condition := SpinFake.M_GetCall(Index := SpinFake.HistoryCount, CallRecord => SpinCall), Message := 'Spin withdrawal must be recorded.');
		AssertTrue(Condition := LiftCWFake.M_GetCall(Index := LiftCWFake.HistoryCount, CallRecord => LiftCWCall), Message := 'Lift CW withdrawal must be recorded.');
		AssertTrue(Condition := LiftCCWFake.M_GetCall(Index := LiftCCWFake.HistoryCount, CallRecord => LiftCCWCall), Message := 'Lift CCW withdrawal must be recorded.');
		AssertTrue(Condition := (SpinCall.Operation = E_FakeAxisOperation.MoveVel)
			AND (LiftCWCall.Operation = E_FakeAxisOperation.MoveVel)
			AND (LiftCCWCall.Operation = E_FakeAxisOperation.MoveVel), Message := 'Natural completion must withdraw MoveVel without issuing Stop.');
		AssertFalse(Condition := SpinCall.Execute OR LiftCWCall.Execute OR LiftCCWCall.Execute, Message := 'Completing must lower every MoveVel request.');
		nSpinHistoryBeforeStop := SpinFake.HistoryCount;
		nLiftCWHistoryBeforeStop := LiftCWFake.HistoryCount;
		nLiftCCWHistoryBeforeStop := LiftCCWFake.HistoryCount;
		nPhase := 7;

	7:
		Ctrl.PackMLIn.eCommand := E_PackMLCommand.Stop;
		Ctrl.PackMLIn.bCommandChangeRequest := TRUE;
		SpinService(Ctrl := Ctrl, Param := SpinParam, Context := Context, Axis_BaseUnit := SpinAxis, ServiceId := 31);
		LiftCWService(Ctrl := Ctrl, Param := LiftCWParam, Context := Context, Axis_BaseUnit := LiftCWAxis, ServiceId := 32);
		LiftCCWService(Ctrl := Ctrl, Param := LiftCCWParam, Context := Context, Axis_BaseUnit := LiftCCWAxis, ServiceId := 33);
		SpinFake.M_CyclicUpdate();
		LiftCWFake.M_CyclicUpdate();
		LiftCCWFake.M_CyclicUpdate();

		AssertTrue(Condition := (SpinService.PackMLOut.eStateCurrent = E_PackMLState.Stopping)
			AND (LiftCWService.PackMLOut.eStateCurrent = E_PackMLState.Stopping)
			AND (LiftCCWService.PackMLOut.eStateCurrent = E_PackMLState.Stopping), Message := 'Stop from Complete must enter Stopping.');
		AssertTrue(Condition := SpinAxis.M_IsResourceOwner(OwnerId := 31)
			AND LiftCWAxis.M_IsResourceOwner(OwnerId := 32)
			AND LiftCCWAxis.M_IsResourceOwner(OwnerId := 33), Message := 'Stopping must retain ownership until physical Stop completes.');
		AssertTrue(Condition := SpinFake.M_GetCall(Index := nSpinHistoryBeforeStop + 2, CallRecord => SpinCall), Message := 'Spin physical Stop request must be recorded.');
		AssertTrue(Condition := LiftCWFake.M_GetCall(Index := nLiftCWHistoryBeforeStop + 2, CallRecord => LiftCWCall), Message := 'Lift CW physical Stop request must be recorded.');
		AssertTrue(Condition := LiftCCWFake.M_GetCall(Index := nLiftCCWHistoryBeforeStop + 2, CallRecord => LiftCCWCall), Message := 'Lift CCW physical Stop request must be recorded.');
		AssertTrue(Condition := (SpinCall.Operation = E_FakeAxisOperation.Stop) AND SpinCall.Accepted AND SpinCall.Execute AND (SpinCall.Deceleration = 13), Message := 'Spin Stop must use the latched Deceleration.');
		AssertTrue(Condition := (LiftCWCall.Operation = E_FakeAxisOperation.Stop) AND LiftCWCall.Accepted AND LiftCWCall.Execute AND (LiftCWCall.Deceleration = 23), Message := 'Lift CW Stop must use the latched Deceleration.');
		AssertTrue(Condition := (LiftCCWCall.Operation = E_FakeAxisOperation.Stop) AND LiftCCWCall.Accepted AND LiftCCWCall.Execute AND (LiftCCWCall.Deceleration = 33), Message := 'Lift CCW Stop must use the latched Deceleration.');
		nPhase := 8;

	8:
		Ctrl.PackMLIn.bCommandChangeRequest := FALSE;
		SpinService(Ctrl := Ctrl, Param := SpinParam, Context := Context, Axis_BaseUnit := SpinAxis, ServiceId := 31);
		LiftCWService(Ctrl := Ctrl, Param := LiftCWParam, Context := Context, Axis_BaseUnit := LiftCWAxis, ServiceId := 32);
		LiftCCWService(Ctrl := Ctrl, Param := LiftCCWParam, Context := Context, Axis_BaseUnit := LiftCCWAxis, ServiceId := 33);
		SpinFake.M_CyclicUpdate();
		LiftCWFake.M_CyclicUpdate();
		LiftCCWFake.M_CyclicUpdate();

		AssertTrue(Condition := (SpinService.PackMLOut.eStateCurrent = E_PackMLState.Stopped)
			AND (LiftCWService.PackMLOut.eStateCurrent = E_PackMLState.Stopped)
			AND (LiftCCWService.PackMLOut.eStateCurrent = E_PackMLState.Stopped), Message := 'Physical Stop completion must reach Stopped.');
		AssertFalse(Condition := SpinAxis.M_IsResourceOwner(OwnerId := 31)
			OR LiftCWAxis.M_IsResourceOwner(OwnerId := 32)
			OR LiftCCWAxis.M_IsResourceOwner(OwnerId := 33), Message := 'Stopped Services must release Axis ownership.');
		AssertTrue(Condition := (SpinService.Status.ErrorList[1].MainErrorId = 0)
			AND (LiftCWService.Status.ErrorList[1].MainErrorId = 0)
			AND (LiftCCWService.Status.ErrorList[1].MainErrorId = 0), Message := 'Successful MoveVel completion and Stop must not create Service errors.');
		AssertFalse(Condition := SpinFake.HistoryOverflowed OR LiftCWFake.HistoryOverflowed OR LiftCCWFake.HistoryOverflowed, Message := 'MoveVel test history must not overflow.');
		nPhase := 0;
		TEST_FINISHED();
END_CASE
END_METHOD

METHOD ResetToIdleKeepsOwnershipUntilStop
VAR_INST
	Axis : I_Axis_BaseUnit;
	Ctrl : ST_ServiceCtrl;
	Param : ST_Chamber1SpinAxisMoveVelParam;
	Context : ST_ServiceContext;
	nPhase : UINT;
END_VAR
TEST('ResetToIdleKeepsOwnershipUntilStop');

CASE nPhase OF
	0:
		ResetFake.M_ResetScenario();
		Axis := ResetFake;
		Param.Velocity := 41;
		Param.Acceleration := 42;
		Param.Deceleration := 43;
		Context.ModuleId := 1;
		AssertTrue(Condition := ResetFake.M_QueueResult(Operation := E_FakeAxisOperation.MoveVel, AfterActiveCycles := 1, Done := FALSE, InVelocity := TRUE, Error := FALSE, ErrorId := 0), Message := 'Reset-path MoveVel script must be accepted.');
		AssertTrue(Condition := ResetFake.M_QueueResult(Operation := E_FakeAxisOperation.Stop, AfterActiveCycles := 1, Done := TRUE, InVelocity := FALSE, Error := FALSE, ErrorId := 0), Message := 'Reset-path Stop script must be accepted.');
		ResetService(Ctrl := Ctrl, Param := Param, Context := Context, Axis_BaseUnit := Axis, ServiceId := 41);
		ResetFake.M_CyclicUpdate();
		AssertTrue(Condition := ResetService.PackMLOut.eStateCurrent = E_PackMLState.Aborted, Message := 'Initial scan must reach Aborted.');
		nPhase := 1;

	1:
		Ctrl.PackMLIn.eCommand := E_PackMLCommand.Clear;
		Ctrl.PackMLIn.bCommandChangeRequest := TRUE;
		ResetService(Ctrl := Ctrl, Param := Param, Context := Context, Axis_BaseUnit := Axis, ServiceId := 41);
		ResetFake.M_CyclicUpdate();
		Ctrl.PackMLIn.bCommandChangeRequest := FALSE;
		ResetService(Ctrl := Ctrl, Param := Param, Context := Context, Axis_BaseUnit := Axis, ServiceId := 41);
		ResetFake.M_CyclicUpdate();
		Ctrl.PackMLIn.eCommand := E_PackMLCommand.Reset;
		Ctrl.PackMLIn.bCommandChangeRequest := TRUE;
		ResetService(Ctrl := Ctrl, Param := Param, Context := Context, Axis_BaseUnit := Axis, ServiceId := 41);
		ResetFake.M_CyclicUpdate();
		AssertTrue(Condition := ResetService.PackMLOut.eStateCurrent = E_PackMLState.Idle, Message := 'Setup Reset must reach Idle.');
		nPhase := 2;

	2:
		Ctrl.PackMLIn.bCommandChangeRequest := FALSE;
		ResetService(Ctrl := Ctrl, Param := Param, Context := Context, Axis_BaseUnit := Axis, ServiceId := 41);
		ResetFake.M_CyclicUpdate();
		Ctrl.PackMLIn.eCommand := E_PackMLCommand.Start;
		Ctrl.PackMLIn.bCommandChangeRequest := TRUE;
		ResetService(Ctrl := Ctrl, Param := Param, Context := Context, Axis_BaseUnit := Axis, ServiceId := 41);
		ResetFake.M_CyclicUpdate();
		AssertTrue(Condition := ResetService.PackMLOut.eStateCurrent = E_PackMLState.Execute, Message := 'Valid Start must reach Execute.');
		nPhase := 3;

	3:
		Ctrl.PackMLIn.bCommandChangeRequest := FALSE;
		ResetService(Ctrl := Ctrl, Param := Param, Context := Context, Axis_BaseUnit := Axis, ServiceId := 41);
		ResetFake.M_CyclicUpdate();
		nPhase := 4;

	4:
		ResetService(Ctrl := Ctrl, Param := Param, Context := Context, Axis_BaseUnit := Axis, ServiceId := 41);
		ResetFake.M_CyclicUpdate();
		AssertTrue(Condition := ResetService.PackMLOut.eStateCurrent = E_PackMLState.Completing, Message := 'InVelocity must reach Completing.');
		nPhase := 5;

	5:
		ResetService(Ctrl := Ctrl, Param := Param, Context := Context, Axis_BaseUnit := Axis, ServiceId := 41);
		ResetFake.M_CyclicUpdate();
		AssertTrue(Condition := ResetService.PackMLOut.eStateCurrent = E_PackMLState.Complete, Message := 'Completing must reach Complete.');
		AssertTrue(Condition := Axis.M_IsResourceOwner(OwnerId := 41), Message := 'Complete must keep ownership before Reset.');
		nPhase := 6;

	6:
		Ctrl.PackMLIn.eCommand := E_PackMLCommand.Reset;
		Ctrl.PackMLIn.bCommandChangeRequest := TRUE;
		ResetService(Ctrl := Ctrl, Param := Param, Context := Context, Axis_BaseUnit := Axis, ServiceId := 41);
		ResetFake.M_CyclicUpdate();
		AssertTrue(Condition := ResetService.PackMLOut.eStateCurrent = E_PackMLState.Idle, Message := 'Reset from Complete must reach Idle without stopping motion.');
		AssertTrue(Condition := Axis.M_IsResourceOwner(OwnerId := 41), Message := 'Idle must retain ownership for the continuing MoveVel motion.');
		AssertFalse(Condition := Axis.M_AcquireResource(OwnerId := 99), Message := 'A different Service must not acquire the moving Axis.');
		nPhase := 7;

	7:
		Ctrl.PackMLIn.bCommandChangeRequest := FALSE;
		ResetService(Ctrl := Ctrl, Param := Param, Context := Context, Axis_BaseUnit := Axis, ServiceId := 41);
		ResetFake.M_CyclicUpdate();
		Ctrl.PackMLIn.eCommand := E_PackMLCommand.Stop;
		Ctrl.PackMLIn.bCommandChangeRequest := TRUE;
		ResetService(Ctrl := Ctrl, Param := Param, Context := Context, Axis_BaseUnit := Axis, ServiceId := 41);
		ResetFake.M_CyclicUpdate();
		AssertTrue(Condition := ResetService.PackMLOut.eStateCurrent = E_PackMLState.Stopping, Message := 'Stop from Idle must start physical stopping.');
		AssertTrue(Condition := Axis.M_IsResourceOwner(OwnerId := 41), Message := 'Stopping from Idle must retain ownership until Done.');
		nPhase := 8;

	8:
		Ctrl.PackMLIn.bCommandChangeRequest := FALSE;
		ResetService(Ctrl := Ctrl, Param := Param, Context := Context, Axis_BaseUnit := Axis, ServiceId := 41);
		ResetFake.M_CyclicUpdate();
		AssertTrue(Condition := ResetService.PackMLOut.eStateCurrent = E_PackMLState.Stopped, Message := 'Stop Done must reach Stopped after Reset-to-Idle.');
		AssertFalse(Condition := Axis.M_IsResourceOwner(OwnerId := 41), Message := 'Stopped must release ownership after Reset-to-Idle.');
		AssertTrue(Condition := ResetService.Status.ErrorList[1].MainErrorId = 0, Message := 'Reset and Stop lifecycle must not create errors.');
		nPhase := 0;
		TEST_FINISHED();
END_CASE
END_METHOD

END_FUNCTION_BLOCK

// ---- Tests/Suites/Modules/FB_Chamber1_ModuleTests.TcPOU
FUNCTION_BLOCK FB_Chamber1_ModuleTests EXTENDS TcUnit.FB_TestSuite
VAR
	// Keep large FB instances at Test Suite scope to avoid Method stack overflow.
	MissingAxisModule : FB_Chamber1_Module;
	MissingAxisFake : FB_FakeAxis_BaseUnit;

	LifecycleModule : FB_Chamber1_Module;
	LifecycleSpinFake : FB_FakeAxis_BaseUnit;
	LifecycleLiftFake : FB_FakeAxis_BaseUnit;

	RoutingModule : FB_Chamber1_Module;
	RoutingSpinFake : FB_FakeAxis_BaseUnit;
	RoutingLiftFake : FB_FakeAxis_BaseUnit;

	StoppingModule : FB_Chamber1_Module;
	StoppingSpinFake : FB_FakeAxis_BaseUnit;
	StoppingLiftFake : FB_FakeAxis_BaseUnit;

	MoveVelStopModule : FB_Chamber1_Module;
	MoveVelStopSpinFake : FB_FakeAxis_BaseUnit;
	MoveVelStopLiftFake : FB_FakeAxis_BaseUnit;

END_VAR

MissingAxisPreventsModuleUpdate();
ModuleClearResetAndAutoStartSynchronizesAllServices();
ExecuteRoutesSelectedServiceControlAndParameters();
ModuleStopOverridesServiceControlAndWaitsForCleanup();
CoordinatorRoutesStopToCompletedMoveVel();

METHOD CoordinatorRoutesStopToCompletedMoveVel
VAR_INST
	SpinAxis : I_Axis_BaseUnit;
	LiftAxis : I_Axis_BaseUnit;
	RuntimeConfig : ST_ModuleRuntimeConfig;
	VariableNodeReader : FB_LinkVariableManager;
	ModuleCtrl : ST_ModuleCtrl;
	ServiceCtrl : ST_Chamber1_ServiceCtrl;
	ServiceParam : ST_Chamber1_ServiceParam;
	SystemContext : ST_SystemContext;
	StopCall : ST_FakeAxisCall;
	nHistoryBeforeStop : UINT;
	nPhase : UINT;
END_VAR
TEST('CoordinatorRoutesStopToCompletedMoveVel');

CASE nPhase OF
	0:
		MoveVelStopSpinFake.M_ResetScenario();
		MoveVelStopLiftFake.M_ResetScenario();
		SpinAxis := MoveVelStopSpinFake;
		LiftAxis := MoveVelStopLiftFake;
		ServiceParam.SpinAxisMoveVelCW.Velocity := 51;
		ServiceParam.SpinAxisMoveVelCW.Acceleration := 52;
		ServiceParam.SpinAxisMoveVelCW.Deceleration := 53;
		AssertTrue(Condition := MoveVelStopSpinFake.M_QueueResult(Operation := E_FakeAxisOperation.MoveVel, AfterActiveCycles := 1, Done := FALSE, InVelocity := TRUE, Error := FALSE, ErrorId := 0), Message := 'Module MoveVel script must be accepted.');
		AssertTrue(Condition := MoveVelStopSpinFake.M_QueueResult(Operation := E_FakeAxisOperation.Stop, AfterActiveCycles := 1, Done := TRUE, InVelocity := FALSE, Error := FALSE, ErrorId := 0), Message := 'Module Stop script must be accepted.');
		MoveVelStopModule(ModuleCtrl := ModuleCtrl, SystemContext := SystemContext, HeartbeatIndex := , RuntimeConfig := RuntimeConfig, VariableNodeReader := VariableNodeReader, ServiceCtrl := ServiceCtrl, ServiceParam := ServiceParam, SpinAxis_BaseUnit := SpinAxis, LiftPinAxis_BaseUnit := LiftAxis);
		nPhase := 1;

	1:
		ModuleCtrl.PackMLIn.eCommand := E_PackMLCommand.Clear;
		ModuleCtrl.PackMLIn.bCommandChangeRequest := TRUE;
		MoveVelStopModule(ModuleCtrl := ModuleCtrl, SystemContext := SystemContext, HeartbeatIndex := , RuntimeConfig := RuntimeConfig, VariableNodeReader := VariableNodeReader, ServiceCtrl := ServiceCtrl, ServiceParam := ServiceParam, SpinAxis_BaseUnit := SpinAxis, LiftPinAxis_BaseUnit := LiftAxis);
		nPhase := 2;

	2:
		ModuleCtrl.PackMLIn.bCommandChangeRequest := FALSE;
		MoveVelStopModule(ModuleCtrl := ModuleCtrl, SystemContext := SystemContext, HeartbeatIndex := , RuntimeConfig := RuntimeConfig, VariableNodeReader := VariableNodeReader, ServiceCtrl := ServiceCtrl, ServiceParam := ServiceParam, SpinAxis_BaseUnit := SpinAxis, LiftPinAxis_BaseUnit := LiftAxis);
		nPhase := 3;

	3:
		ModuleCtrl.PackMLIn.eCommand := E_PackMLCommand.Reset;
		ModuleCtrl.PackMLIn.bCommandChangeRequest := TRUE;
		MoveVelStopModule(ModuleCtrl := ModuleCtrl, SystemContext := SystemContext, HeartbeatIndex := , RuntimeConfig := RuntimeConfig, VariableNodeReader := VariableNodeReader, ServiceCtrl := ServiceCtrl, ServiceParam := ServiceParam, SpinAxis_BaseUnit := SpinAxis, LiftPinAxis_BaseUnit := LiftAxis);
		nPhase := 4;

	4:
		ModuleCtrl.PackMLIn.bCommandChangeRequest := FALSE;
		MoveVelStopModule(ModuleCtrl := ModuleCtrl, SystemContext := SystemContext, HeartbeatIndex := , RuntimeConfig := RuntimeConfig, VariableNodeReader := VariableNodeReader, ServiceCtrl := ServiceCtrl, ServiceParam := ServiceParam, SpinAxis_BaseUnit := SpinAxis, LiftPinAxis_BaseUnit := LiftAxis);
		nPhase := 5;

	5:
		MoveVelStopModule(ModuleCtrl := ModuleCtrl, SystemContext := SystemContext, HeartbeatIndex := , RuntimeConfig := RuntimeConfig, VariableNodeReader := VariableNodeReader, ServiceCtrl := ServiceCtrl, ServiceParam := ServiceParam, SpinAxis_BaseUnit := SpinAxis, LiftPinAxis_BaseUnit := LiftAxis);
		nPhase := 6;

	6:
		MoveVelStopModule(ModuleCtrl := ModuleCtrl, SystemContext := SystemContext, HeartbeatIndex := , RuntimeConfig := RuntimeConfig, VariableNodeReader := VariableNodeReader, ServiceCtrl := ServiceCtrl, ServiceParam := ServiceParam, SpinAxis_BaseUnit := SpinAxis, LiftPinAxis_BaseUnit := LiftAxis);
		AssertTrue(Condition := MoveVelStopModule.PackMLOut.eStateCurrent = E_PackMLState.Execute, Message := 'Test setup must bring Module to Execute.');
		nPhase := 7;

	7:
		ServiceCtrl.SpinAxisMoveVelCW.RequestId := 5101;
		ServiceCtrl.SpinAxisMoveVelCW.PackMLIn.eCommand := E_PackMLCommand.Start;
		ServiceCtrl.SpinAxisMoveVelCW.PackMLIn.bCommandChangeRequest := TRUE;
		MoveVelStopModule(ModuleCtrl := ModuleCtrl, SystemContext := SystemContext, HeartbeatIndex := , RuntimeConfig := RuntimeConfig, VariableNodeReader := VariableNodeReader, ServiceCtrl := ServiceCtrl, ServiceParam := ServiceParam, SpinAxis_BaseUnit := SpinAxis, LiftPinAxis_BaseUnit := LiftAxis);
		AssertTrue(Condition := MoveVelStopModule.ServiceStatus.SpinAxisMoveVelCW.PackMLOut.eStateCurrent = E_PackMLState.Execute, Message := 'Coordinator must route upper Start to MoveVel.');
		AssertTrue(Condition := MoveVelStopModule.ServiceStatus.SpinAxisMoveVelCW.ResponseId = 5101, Message := 'MoveVel must acknowledge upper Start RequestId.');
		nPhase := 8;

	8:
		ServiceCtrl.SpinAxisMoveVelCW.PackMLIn.bCommandChangeRequest := FALSE;
		MoveVelStopModule(ModuleCtrl := ModuleCtrl, SystemContext := SystemContext, HeartbeatIndex := , RuntimeConfig := RuntimeConfig, VariableNodeReader := VariableNodeReader, ServiceCtrl := ServiceCtrl, ServiceParam := ServiceParam, SpinAxis_BaseUnit := SpinAxis, LiftPinAxis_BaseUnit := LiftAxis);
		nPhase := 9;

	9:
		MoveVelStopModule(ModuleCtrl := ModuleCtrl, SystemContext := SystemContext, HeartbeatIndex := , RuntimeConfig := RuntimeConfig, VariableNodeReader := VariableNodeReader, ServiceCtrl := ServiceCtrl, ServiceParam := ServiceParam, SpinAxis_BaseUnit := SpinAxis, LiftPinAxis_BaseUnit := LiftAxis);
		AssertTrue(Condition := MoveVelStopModule.ServiceStatus.SpinAxisMoveVelCW.PackMLOut.eStateCurrent = E_PackMLState.Completing, Message := 'InVelocity must move the routed Service to Completing.');
		nPhase := 10;

	10:
		MoveVelStopModule(ModuleCtrl := ModuleCtrl, SystemContext := SystemContext, HeartbeatIndex := , RuntimeConfig := RuntimeConfig, VariableNodeReader := VariableNodeReader, ServiceCtrl := ServiceCtrl, ServiceParam := ServiceParam, SpinAxis_BaseUnit := SpinAxis, LiftPinAxis_BaseUnit := LiftAxis);
		AssertTrue(Condition := MoveVelStopModule.ServiceStatus.SpinAxisMoveVelCW.PackMLOut.eStateCurrent = E_PackMLState.Complete, Message := 'MoveVel must reach Complete after withdrawing its request.');
		AssertTrue(Condition := SpinAxis.M_IsResourceOwner(OwnerId := E_Chamber1ServiceId.SpinAxisMoveVelCW), Message := 'Completed MoveVel must still own Spin Axis.');
		nHistoryBeforeStop := MoveVelStopSpinFake.HistoryCount;
		nPhase := 11;

	11:
		ServiceCtrl.SpinAxisMoveVelCW.RequestId := 5102;
		ServiceCtrl.SpinAxisMoveVelCW.PackMLIn.eCommand := E_PackMLCommand.Stop;
		ServiceCtrl.SpinAxisMoveVelCW.PackMLIn.bCommandChangeRequest := TRUE;
		MoveVelStopModule(ModuleCtrl := ModuleCtrl, SystemContext := SystemContext, HeartbeatIndex := , RuntimeConfig := RuntimeConfig, VariableNodeReader := VariableNodeReader, ServiceCtrl := ServiceCtrl, ServiceParam := ServiceParam, SpinAxis_BaseUnit := SpinAxis, LiftPinAxis_BaseUnit := LiftAxis);
		AssertTrue(Condition := MoveVelStopModule.ServiceStatus.SpinAxisMoveVelCW.PackMLOut.eStateCurrent = E_PackMLState.Stopping, Message := 'Coordinator must route upper Stop from Complete.');
		AssertTrue(Condition := MoveVelStopModule.ServiceStatus.SpinAxisMoveVelCW.ResponseId = 5102, Message := 'MoveVel must acknowledge upper Stop RequestId.');
		AssertTrue(Condition := MoveVelStopSpinFake.M_GetCall(Index := nHistoryBeforeStop + 2, CallRecord => StopCall), Message := 'Routed physical Stop must be recorded.');
		AssertTrue(Condition := (StopCall.Operation = E_FakeAxisOperation.Stop) AND StopCall.Accepted AND StopCall.Execute AND (StopCall.Deceleration = 53), Message := 'Routed Stop must execute with the latched Deceleration.');
		nPhase := 12;

	12:
		ServiceCtrl.SpinAxisMoveVelCW.PackMLIn.bCommandChangeRequest := FALSE;
		MoveVelStopModule(ModuleCtrl := ModuleCtrl, SystemContext := SystemContext, HeartbeatIndex := , RuntimeConfig := RuntimeConfig, VariableNodeReader := VariableNodeReader, ServiceCtrl := ServiceCtrl, ServiceParam := ServiceParam, SpinAxis_BaseUnit := SpinAxis, LiftPinAxis_BaseUnit := LiftAxis);
		AssertTrue(Condition := MoveVelStopModule.ServiceStatus.SpinAxisMoveVelCW.PackMLOut.eStateCurrent = E_PackMLState.Stopped, Message := 'Physical Stop Done must reach Stopped through Coordinator.');
		AssertFalse(Condition := SpinAxis.M_IsResourceOwner(OwnerId := E_Chamber1ServiceId.SpinAxisMoveVelCW), Message := 'Routed Stop completion must release Spin Axis.');
		nPhase := 0;
		TEST_FINISHED();
END_CASE
END_METHOD

METHOD ExecuteRoutesSelectedServiceControlAndParameters
VAR_INST
	SpinAxis : I_Axis_BaseUnit;
	LiftAxis : I_Axis_BaseUnit;
	HwInput : ST_Chamber1_Signal_In;
	HwOutput : ST_Chamber1_Signal_Out;
	RuntimeConfig : ST_ModuleRuntimeConfig;
	VariableNodeReader : FB_LinkVariableManager;
	ModuleCtrl : ST_ModuleCtrl;
	ServiceCtrl : ST_Chamber1_ServiceCtrl;
	ServiceParam : ST_Chamber1_ServiceParam;
	SystemContext : ST_SystemContext;
	CallRecord : ST_FakeAxisCall;
	nPhase : UINT;
END_VAR
TEST('ExecuteRoutesSelectedServiceControlAndParameters');

CASE nPhase OF
	0:
		// Set Module dependencies and selected Service param
		RoutingSpinFake.M_ResetScenario();
		RoutingLiftFake.M_ResetScenario();
		SpinAxis := RoutingSpinFake;
		LiftAxis := RoutingLiftFake;
		SystemContext.UtcDateTime := '20260813123456007';
		ServiceParam.SpinAxisMoveAbs.Position := 125.25;
		ServiceParam.SpinAxisMoveAbs.Velocity := 15;
		ServiceParam.SpinAxisMoveAbs.Acceleration := 25;
		ServiceParam.SpinAxisMoveAbs.Deceleration := 35;

		// Initial Module scan
		RoutingModule(
			ModuleCtrl:= ModuleCtrl,
			SystemContext:= SystemContext,
			HeartbeatIndex:= ,
			RuntimeConfig:= RuntimeConfig,
			VariableNodeReader:= VariableNodeReader,
			ServiceCtrl:= ServiceCtrl,
			ServiceParam:= ServiceParam,
			SpinAxis_BaseUnit:= SpinAxis,
			LiftPinAxis_BaseUnit:= LiftAxis);

		AssertTrue(
			Condition := (RoutingModule.ServiceStatus.SpinAxisMoveAbs.CompletionBehavior = E_ServiceCompletionBehavior.NaturalCompletion)
				AND (RoutingModule.ServiceStatus.LiftPinAxisMoveAbs.CompletionBehavior = E_ServiceCompletionBehavior.NaturalCompletion)
				AND (RoutingModule.ServiceStatus.SpinAxisMoveVelCW.CompletionBehavior = E_ServiceCompletionBehavior.NaturalCompletion)
				AND (RoutingModule.ServiceStatus.LiftPinAxisMoveVelCW.CompletionBehavior = E_ServiceCompletionBehavior.NaturalCompletion)
				AND (RoutingModule.ServiceStatus.LiftPinAxisMoveVelCCW.CompletionBehavior = E_ServiceCompletionBehavior.NaturalCompletion)
				AND (RoutingModule.ServiceStatus.PreparePosition.CompletionBehavior = E_ServiceCompletionBehavior.NaturalCompletion),
			Message := 'Finite Chamber1 Services must publish NaturalCompletion on their first cyclic update.');
		AssertTrue(
			Condition := RoutingModule.ServiceStatus.SpinAxisJogCW.CompletionBehavior = E_ServiceCompletionBehavior.ExecuteUntilExternalStop,
			Message := 'SpinAxisJogCW must remain the continuous Chamber1 Service.');
		nPhase := 1;

	1:
		// Clear Module and Services
		ModuleCtrl.PackMLIn.eCommand := E_PackMLCommand.Clear;
		ModuleCtrl.PackMLIn.bCommandChangeRequest := TRUE;
		RoutingModule(
			ModuleCtrl:= ModuleCtrl, 
			SystemContext:= SystemContext, 
			HeartbeatIndex:= , 
			RuntimeConfig:= RuntimeConfig, 
			VariableNodeReader:= VariableNodeReader,  
			ServiceCtrl:= ServiceCtrl, 
			ServiceParam:= ServiceParam, 
			SpinAxis_BaseUnit:= SpinAxis, 
			LiftPinAxis_BaseUnit:= LiftAxis);
			nPhase := 2;

	2:
		// Finish Clearing
		ModuleCtrl.PackMLIn.bCommandChangeRequest := FALSE;
		RoutingModule(
			ModuleCtrl:= ModuleCtrl, 
			SystemContext:= SystemContext, 
			HeartbeatIndex:= , 
			RuntimeConfig:= RuntimeConfig, 
			VariableNodeReader:= VariableNodeReader,  
			ServiceCtrl:= ServiceCtrl, 
			ServiceParam:= ServiceParam, 
			SpinAxis_BaseUnit:= SpinAxis, 
			LiftPinAxis_BaseUnit:= LiftAxis);
		nPhase := 3;

	3:
		// Reset Module and Services
		ModuleCtrl.PackMLIn.eCommand := E_PackMLCommand.Reset;
		ModuleCtrl.PackMLIn.bCommandChangeRequest := TRUE;
		RoutingModule(
			ModuleCtrl:= ModuleCtrl, 
			SystemContext:= SystemContext, 
			HeartbeatIndex:= , 
			RuntimeConfig:= RuntimeConfig, 
			VariableNodeReader:= VariableNodeReader,  
			ServiceCtrl:= ServiceCtrl, 
			ServiceParam:= ServiceParam, 
			SpinAxis_BaseUnit:= SpinAxis, 
			LiftPinAxis_BaseUnit:= LiftAxis);
		nPhase := 4;

	4:
		// Finish Resetting
		ModuleCtrl.PackMLIn.bCommandChangeRequest := FALSE;
		RoutingModule(
			ModuleCtrl:= ModuleCtrl, 
			SystemContext:= SystemContext, 
			HeartbeatIndex:= , 
			RuntimeConfig:= RuntimeConfig, 
			VariableNodeReader:= VariableNodeReader,  
			ServiceCtrl:= ServiceCtrl, 
			ServiceParam:= ServiceParam, 
			SpinAxis_BaseUnit:= SpinAxis, 
			LiftPinAxis_BaseUnit:= LiftAxis);
		nPhase := 5;

	5:
		// Queue Module automatic Start
		RoutingModule(
			ModuleCtrl:= ModuleCtrl, 
			SystemContext:= SystemContext, 
			HeartbeatIndex:= , 
			RuntimeConfig:= RuntimeConfig, 
			VariableNodeReader:= VariableNodeReader,  
			ServiceCtrl:= ServiceCtrl, 
			ServiceParam:= ServiceParam, 
			SpinAxis_BaseUnit:= SpinAxis, 
			LiftPinAxis_BaseUnit:= LiftAxis);
		nPhase := 6;

	6:
		// Process Module automatic Start
		RoutingModule(
			ModuleCtrl:= ModuleCtrl, 
			SystemContext:= SystemContext, 
			HeartbeatIndex:= , 
			RuntimeConfig:= RuntimeConfig, 
			VariableNodeReader:= VariableNodeReader,  
			ServiceCtrl:= ServiceCtrl, 
			ServiceParam:= ServiceParam, 
			SpinAxis_BaseUnit:= SpinAxis, 
			LiftPinAxis_BaseUnit:= LiftAxis);
		AssertTrue(Condition := RoutingModule.PackMLOut.eStateCurrent = E_PackMLState.Execute, Message := 'Test setup must bring the Module to Execute.');
		nPhase := 7;

	7:
		// Start only SpinAxisMoveAbs through external ServiceCtrl
		ServiceCtrl.SpinAxisMoveAbs.RequestId := 2001;
		ServiceCtrl.SpinAxisMoveAbs.PackMLIn.eCommand := E_PackMLCommand.Start;
		ServiceCtrl.SpinAxisMoveAbs.PackMLIn.bCommandChangeRequest := TRUE;
		RoutingModule(
			ModuleCtrl:= ModuleCtrl, 
			SystemContext:= SystemContext, 
			HeartbeatIndex:= , 
			RuntimeConfig:= RuntimeConfig, 
			VariableNodeReader:= VariableNodeReader,  
			ServiceCtrl:= ServiceCtrl, 
			ServiceParam:= ServiceParam, 
			SpinAxis_BaseUnit:= SpinAxis, 
			LiftPinAxis_BaseUnit:= LiftAxis);
			
		// Only the selected Service may enter Execute and own Spin Axis
		AssertTrue(Condition := RoutingModule.ServiceStatus.SpinAxisMoveAbs.PackMLOut.eStateCurrent = E_PackMLState.Execute, Message := 'External Start must route to SpinAxisMoveAbs.');
		AssertTrue(Condition := RoutingModule.ServiceStatus.SpinAxisMoveAbs.ResponseId = 2001, Message := 'Selected Service must acknowledge its RequestId.');
		AssertTrue(Condition := SpinAxis.M_IsResourceOwner(OwnerId := E_Chamber1ServiceId.SpinAxisMoveAbs), Message := 'SpinAxisMoveAbs must acquire Spin Axis with its assigned OwnerId.');
		AssertTrue(
			Condition := (RoutingModule.ServiceStatus.SpinAxisMoveAbs.CompletionBehavior = E_ServiceCompletionBehavior.NaturalCompletion)
				AND (RoutingModule.ServiceStatus.LiftPinAxisMoveAbs.CompletionBehavior = E_ServiceCompletionBehavior.NaturalCompletion)
				AND (RoutingModule.ServiceStatus.SpinAxisMoveVelCW.CompletionBehavior = E_ServiceCompletionBehavior.NaturalCompletion)
				AND (RoutingModule.ServiceStatus.LiftPinAxisMoveVelCW.CompletionBehavior = E_ServiceCompletionBehavior.NaturalCompletion)
				AND (RoutingModule.ServiceStatus.LiftPinAxisMoveVelCCW.CompletionBehavior = E_ServiceCompletionBehavior.NaturalCompletion)
				AND (RoutingModule.ServiceStatus.PreparePosition.CompletionBehavior = E_ServiceCompletionBehavior.NaturalCompletion)
				AND (RoutingModule.ServiceStatus.SpinAxisJogCW.CompletionBehavior = E_ServiceCompletionBehavior.ExecuteUntilExternalStop),
			Message := 'Completion behavior must remain stable after Module and Service state transitions.');
		AssertTrue(
			Condition := (RoutingModule.ServiceStatus.SpinAxisJogCW.PackMLOut.eStateCurrent = E_PackMLState.Idle)
				AND (RoutingModule.ServiceStatus.SpinAxisMoveVelCW.PackMLOut.eStateCurrent = E_PackMLState.Idle)
				AND (RoutingModule.ServiceStatus.LiftPinAxisMoveVelCW.PackMLOut.eStateCurrent = E_PackMLState.Idle)
				AND (RoutingModule.ServiceStatus.LiftPinAxisMoveVelCCW.PackMLOut.eStateCurrent = E_PackMLState.Idle)
				AND (RoutingModule.ServiceStatus.LiftPinAxisMoveAbs.PackMLOut.eStateCurrent = E_PackMLState.Idle),
			Message := 'Unselected Services must remain Idle.');
		AssertTrue(Condition := RoutingLiftFake.HistoryCount = 0, Message := 'Selected Spin Service must not issue a LiftPin Axis command.');
		nPhase := 8;

	8:
		// Reset Service request flag and execute MoveAbs
		ServiceCtrl.SpinAxisMoveAbs.PackMLIn.bCommandChangeRequest := FALSE;
		RoutingModule(
			ModuleCtrl:= ModuleCtrl, 
			SystemContext:= SystemContext, 
			HeartbeatIndex:= , 
			RuntimeConfig:= RuntimeConfig, 
			VariableNodeReader:= VariableNodeReader,  
			ServiceCtrl:= ServiceCtrl, 
			ServiceParam:= ServiceParam, 
			SpinAxis_BaseUnit:= SpinAxis, 
			LiftPinAxis_BaseUnit:= LiftAxis);
			
		// Check OwnerId and all parameters passed through Module
		AssertTrue(Condition := RoutingSpinFake.M_GetCall(Index := RoutingSpinFake.HistoryCount, CallRecord => CallRecord), Message := 'Module-routed MoveAbs command must be recorded.');
		AssertTrue(Condition := CallRecord.Operation = E_FakeAxisOperation.MoveAbs, Message := 'Selected Service must issue MoveAbs.');
		AssertTrue(Condition := CallRecord.Accepted AND CallRecord.Execute, Message := 'Selected MoveAbs command must be active and accepted.');
		AssertTrue(Condition := CallRecord.OwnerId = E_Chamber1ServiceId.SpinAxisMoveAbs, Message := 'MoveAbs command must use the assigned Service OwnerId.');
		AssertTrue(Condition := CallRecord.Position = ServiceParam.SpinAxisMoveAbs.Position, Message := 'Module must pass Position unchanged.');
		AssertTrue(Condition := CallRecord.Velocity = ServiceParam.SpinAxisMoveAbs.Velocity, Message := 'Module must pass Velocity unchanged.');
		AssertTrue(Condition := CallRecord.Acceleration = ServiceParam.SpinAxisMoveAbs.Acceleration, Message := 'Module must pass Acceleration unchanged.');
		AssertTrue(Condition := CallRecord.Deceleration = ServiceParam.SpinAxisMoveAbs.Deceleration, Message := 'Module must pass Deceleration unchanged.');
		AssertTrue(Condition := RoutingLiftFake.HistoryCount = 0, Message := 'Routing selected Spin Service must leave LiftPin Axis untouched.');
		nPhase := 0;

		TEST_FINISHED();
END_CASE
END_METHOD

METHOD MissingAxisPreventsModuleUpdate
VAR_INST
	BoundAxis : I_Axis_BaseUnit;
	UnboundAxis : I_Axis_BaseUnit;
	SpinAxis : I_Axis_BaseUnit;
	LiftAxis : I_Axis_BaseUnit;
	HwInput : ST_Chamber1_Signal_In;
	HwOutput : ST_Chamber1_Signal_Out;
	RuntimeConfig : ST_ModuleRuntimeConfig;
	VariableNodeReader : FB_LinkVariableManager;
	ModuleCtrl : ST_ModuleCtrl;
	ServiceCtrl : ST_Chamber1_ServiceCtrl;
	ServiceParam : ST_Chamber1_ServiceParam;
	SystemContext : ST_SystemContext;
	nPhase : UINT;
END_VAR
TEST('MissingAxisPreventsModuleUpdate');

CASE nPhase OF
	0:
		// Bind Spin Axis only
		MissingAxisFake.M_ResetScenario();
		BoundAxis := MissingAxisFake;
		SpinAxis := BoundAxis;
		LiftAxis := UnboundAxis;

		// Cyclic update
		MissingAxisModule(
			ModuleCtrl:= ModuleCtrl,
			SystemContext:= SystemContext,
			HeartbeatIndex:= ,
			RuntimeConfig:= RuntimeConfig,
			VariableNodeReader:= VariableNodeReader,
			ServiceCtrl:= ServiceCtrl,
			ServiceParam:= ServiceParam,
			SpinAxis_BaseUnit:= SpinAxis,
			LiftPinAxis_BaseUnit:= LiftAxis);

		// Missing LiftPin Axis must prevent the entire Module update
		AssertTrue(Condition := MissingAxisModule.PackMLOut.eStateCurrent = E_PackMLState.Undefined, Message := 'Missing LiftPin Axis must keep the Module Undefined.');
		AssertTrue(Condition := MissingAxisFake.CurrentCycle = 0, Message := 'Missing LiftPin Axis must prevent Spin Axis cyclic update.');
		AssertTrue(Condition := MissingAxisFake.HistoryCount = 0, Message := 'Missing LiftPin Axis must prevent Axis commands.');
		AssertTrue(
			Condition := (MissingAxisModule.ServiceStatus.SpinAxisJogCW.PackMLOut.eStateCurrent = E_PackMLState.Undefined)
				AND (MissingAxisModule.ServiceStatus.SpinAxisMoveAbs.PackMLOut.eStateCurrent = E_PackMLState.Undefined)
				AND (MissingAxisModule.ServiceStatus.SpinAxisMoveVelCW.PackMLOut.eStateCurrent = E_PackMLState.Undefined)
				AND (MissingAxisModule.ServiceStatus.LiftPinAxisMoveVelCW.PackMLOut.eStateCurrent = E_PackMLState.Undefined)
				AND (MissingAxisModule.ServiceStatus.LiftPinAxisMoveVelCCW.PackMLOut.eStateCurrent = E_PackMLState.Undefined)
				AND (MissingAxisModule.ServiceStatus.LiftPinAxisMoveAbs.PackMLOut.eStateCurrent = E_PackMLState.Undefined),
			Message := 'Missing LiftPin Axis must prevent every Service update.');
		AssertTrue(
			Condition := (MissingAxisModule.ServiceStatus.SpinAxisJogCW.CompletionBehavior = E_ServiceCompletionBehavior.Unknown)
				AND (MissingAxisModule.ServiceStatus.SpinAxisMoveAbs.CompletionBehavior = E_ServiceCompletionBehavior.Unknown)
				AND (MissingAxisModule.ServiceStatus.SpinAxisMoveVelCW.CompletionBehavior = E_ServiceCompletionBehavior.Unknown)
				AND (MissingAxisModule.ServiceStatus.LiftPinAxisMoveVelCW.CompletionBehavior = E_ServiceCompletionBehavior.Unknown)
				AND (MissingAxisModule.ServiceStatus.LiftPinAxisMoveVelCCW.CompletionBehavior = E_ServiceCompletionBehavior.Unknown)
				AND (MissingAxisModule.ServiceStatus.LiftPinAxisMoveAbs.CompletionBehavior = E_ServiceCompletionBehavior.Unknown),
			Message := 'Services that have not run a cyclic update must keep Unknown completion behavior.');
		nPhase := 1;

	1:
		// Bind LiftPin Axis only
		SpinAxis := UnboundAxis;
		LiftAxis := BoundAxis;

		// Cyclic update
		MissingAxisModule(
			ModuleCtrl:= ModuleCtrl,
			SystemContext:= SystemContext,
			HeartbeatIndex:= ,
			RuntimeConfig:= RuntimeConfig,
			VariableNodeReader:= VariableNodeReader,
			ServiceCtrl:= ServiceCtrl,
			ServiceParam:= ServiceParam,
			SpinAxis_BaseUnit:= SpinAxis,
			LiftPinAxis_BaseUnit:= LiftAxis);

		// Missing Spin Axis must prevent the entire Module update
		AssertTrue(Condition := MissingAxisModule.PackMLOut.eStateCurrent = E_PackMLState.Undefined, Message := 'Missing Spin Axis must keep the Module Undefined.');
		AssertTrue(Condition := MissingAxisFake.CurrentCycle = 0, Message := 'Missing Spin Axis must prevent LiftPin Axis cyclic update.');
		AssertTrue(Condition := MissingAxisFake.HistoryCount = 0, Message := 'Missing Spin Axis must prevent Axis commands.');
		nPhase := 0;

		TEST_FINISHED();
END_CASE
END_METHOD

METHOD ModuleClearResetAndAutoStartSynchronizesAllServices
VAR_INST
	SpinAxis : I_Axis_BaseUnit;
	LiftAxis : I_Axis_BaseUnit;
	HwInput : ST_Chamber1_Signal_In;
	HwOutput : ST_Chamber1_Signal_Out;
	RuntimeConfig : ST_ModuleRuntimeConfig;
	VariableNodeReader : FB_LinkVariableManager;
	ModuleCtrl : ST_ModuleCtrl;
	ServiceCtrl : ST_Chamber1_ServiceCtrl;
	ServiceParam : ST_Chamber1_ServiceParam;
	SystemContext : ST_SystemContext;
	nPhase : UINT;
END_VAR
TEST('ModuleClearResetAndAutoStartSynchronizesAllServices');

CASE nPhase OF
	0:
		// Set Module dependencies
		LifecycleSpinFake.M_ResetScenario();
		LifecycleLiftFake.M_ResetScenario();
		SpinAxis := LifecycleSpinFake;
		LiftAxis := LifecycleLiftFake;
		SystemContext.UtcDateTime := '20260813123456007';

		// 1st Module scan
		LifecycleModule(
			ModuleCtrl:= ModuleCtrl,
			SystemContext:= SystemContext,
			HeartbeatIndex:= ,
			RuntimeConfig:= RuntimeConfig,
			VariableNodeReader:= VariableNodeReader,
			ServiceCtrl:= ServiceCtrl,
			ServiceParam:= ServiceParam,
			SpinAxis_BaseUnit:= SpinAxis,
			LiftPinAxis_BaseUnit:= LiftAxis);

		// Module and every Service leave Undefined together
		AssertTrue(Condition := LifecycleModule.PackMLOut.eStateCurrent = E_PackMLState.Aborted, Message := 'Initial Module scan must reach Aborted.');
		AssertTrue(
			Condition := (LifecycleModule.ServiceStatus.SpinAxisJogCW.PackMLOut.eStateCurrent = E_PackMLState.Aborted)
				AND (LifecycleModule.ServiceStatus.SpinAxisMoveAbs.PackMLOut.eStateCurrent = E_PackMLState.Aborted)
				AND (LifecycleModule.ServiceStatus.SpinAxisMoveVelCW.PackMLOut.eStateCurrent = E_PackMLState.Aborted)
				AND (LifecycleModule.ServiceStatus.LiftPinAxisMoveVelCW.PackMLOut.eStateCurrent = E_PackMLState.Aborted)
				AND (LifecycleModule.ServiceStatus.LiftPinAxisMoveVelCCW.PackMLOut.eStateCurrent = E_PackMLState.Aborted)
				AND (LifecycleModule.ServiceStatus.LiftPinAxisMoveAbs.PackMLOut.eStateCurrent = E_PackMLState.Aborted),
			Message := 'Initial scan must route every Service to Aborted.');
		AssertTrue(Condition := (LifecycleSpinFake.CurrentCycle = 1) AND (LifecycleLiftFake.CurrentCycle = 1), Message := 'Module must update each BaseUnit exactly once per scan.');
		nPhase := 1;

	1:
		// Set Module PackML cmd: Clear
		ModuleCtrl.RequestId := 1001;
		ModuleCtrl.PackMLIn.eCommand := E_PackMLCommand.Clear;
		ModuleCtrl.PackMLIn.bCommandChangeRequest := TRUE;

		// Cyclic update
		LifecycleModule(
			ModuleCtrl:= ModuleCtrl,
			SystemContext:= SystemContext,
			HeartbeatIndex:= ,
			RuntimeConfig:= RuntimeConfig,
			VariableNodeReader:= VariableNodeReader,
			ServiceCtrl:= ServiceCtrl,
			ServiceParam:= ServiceParam,
			SpinAxis_BaseUnit:= SpinAxis,
			LiftPinAxis_BaseUnit:= LiftAxis);

		// Module waits one scan for all ServiceStatus values
		AssertTrue(Condition := LifecycleModule.PackMLOut.eStateCurrent = E_PackMLState.Clearing, Message := 'Module must remain Clearing while Services process Clear.');
		AssertTrue(
			Condition := (LifecycleModule.ServiceStatus.SpinAxisJogCW.PackMLOut.eStateCurrent = E_PackMLState.Stopped)
				AND (LifecycleModule.ServiceStatus.SpinAxisMoveAbs.PackMLOut.eStateCurrent = E_PackMLState.Stopped)
				AND (LifecycleModule.ServiceStatus.SpinAxisMoveVelCW.PackMLOut.eStateCurrent = E_PackMLState.Stopped)
				AND (LifecycleModule.ServiceStatus.LiftPinAxisMoveVelCW.PackMLOut.eStateCurrent = E_PackMLState.Stopped)
				AND (LifecycleModule.ServiceStatus.LiftPinAxisMoveVelCCW.PackMLOut.eStateCurrent = E_PackMLState.Stopped)
				AND (LifecycleModule.ServiceStatus.LiftPinAxisMoveAbs.PackMLOut.eStateCurrent = E_PackMLState.Stopped),
			Message := 'Module Clear must route every Service to Stopped.');
		AssertTrue(Condition := LifecycleModule.ModuleStatus.ResponseId = 1001, Message := 'Module must acknowledge the Clear RequestId.');
		nPhase := 2;

	2:
		// Reset request flag
		ModuleCtrl.PackMLIn.bCommandChangeRequest := FALSE;

		// Cyclic update
		LifecycleModule(
			ModuleCtrl:= ModuleCtrl,
			SystemContext:= SystemContext,
			HeartbeatIndex:= ,
			RuntimeConfig:= RuntimeConfig,
			VariableNodeReader:= VariableNodeReader,
			ServiceCtrl:= ServiceCtrl,
			ServiceParam:= ServiceParam,
			SpinAxis_BaseUnit:= SpinAxis,
			LiftPinAxis_BaseUnit:= LiftAxis);

		// Module completes Clearing only after observing all Services Stopped
		AssertTrue(Condition := LifecycleModule.PackMLOut.eStateCurrent = E_PackMLState.Stopped, Message := 'Module must reach Stopped after every Service is Stopped.');
		nPhase := 3;

	3:
		// Set Module PackML cmd: Reset
		ModuleCtrl.RequestId := 1002;
		ModuleCtrl.PackMLIn.eCommand := E_PackMLCommand.Reset;
		ModuleCtrl.PackMLIn.bCommandChangeRequest := TRUE;

		// Cyclic update
		LifecycleModule(
			ModuleCtrl:= ModuleCtrl,
			SystemContext:= SystemContext,
			HeartbeatIndex:= ,
			RuntimeConfig:= RuntimeConfig,
			VariableNodeReader:= VariableNodeReader,
			ServiceCtrl:= ServiceCtrl,
			ServiceParam:= ServiceParam,
			SpinAxis_BaseUnit:= SpinAxis,
			LiftPinAxis_BaseUnit:= LiftAxis);

		// Module waits one scan for all ServiceStatus values
		AssertTrue(Condition := LifecycleModule.PackMLOut.eStateCurrent = E_PackMLState.Resetting, Message := 'Module must remain Resetting while Services process Reset.');
		AssertTrue(
			Condition := (LifecycleModule.ServiceStatus.SpinAxisJogCW.PackMLOut.eStateCurrent = E_PackMLState.Idle)
				AND (LifecycleModule.ServiceStatus.SpinAxisMoveAbs.PackMLOut.eStateCurrent = E_PackMLState.Idle)
				AND (LifecycleModule.ServiceStatus.SpinAxisMoveVelCW.PackMLOut.eStateCurrent = E_PackMLState.Idle)
				AND (LifecycleModule.ServiceStatus.LiftPinAxisMoveVelCW.PackMLOut.eStateCurrent = E_PackMLState.Idle)
				AND (LifecycleModule.ServiceStatus.LiftPinAxisMoveVelCCW.PackMLOut.eStateCurrent = E_PackMLState.Idle)
				AND (LifecycleModule.ServiceStatus.LiftPinAxisMoveAbs.PackMLOut.eStateCurrent = E_PackMLState.Idle),
			Message := 'Module Reset must route every Service to Idle.');
		AssertTrue(Condition := LifecycleModule.ModuleStatus.ResponseId = 1002, Message := 'Module must acknowledge the Reset RequestId.');
		nPhase := 4;

	4:
		// Reset request flag
		ModuleCtrl.PackMLIn.bCommandChangeRequest := FALSE;

		// Cyclic update
		LifecycleModule(
			ModuleCtrl:= ModuleCtrl,
			SystemContext:= SystemContext,
			HeartbeatIndex:= ,
			RuntimeConfig:= RuntimeConfig,
			VariableNodeReader:= VariableNodeReader,
			ServiceCtrl:= ServiceCtrl,
			ServiceParam:= ServiceParam,
			SpinAxis_BaseUnit:= SpinAxis,
			LiftPinAxis_BaseUnit:= LiftAxis);

		// Module completes Resetting only after observing all Services Idle
		AssertTrue(Condition := LifecycleModule.PackMLOut.eStateCurrent = E_PackMLState.Idle, Message := 'Module must reach Idle after every Service is Idle.');
		nPhase := 5;

	5:
		// Idle hook queues an internal Start command
		LifecycleModule(
			ModuleCtrl:= ModuleCtrl,
			SystemContext:= SystemContext,
			HeartbeatIndex:= ,
			RuntimeConfig:= RuntimeConfig,
			VariableNodeReader:= VariableNodeReader,
			ServiceCtrl:= ServiceCtrl,
			ServiceParam:= ServiceParam,
			SpinAxis_BaseUnit:= SpinAxis,
			LiftPinAxis_BaseUnit:= LiftAxis);

		AssertTrue(Condition := LifecycleModule.PackMLOut.eStateCurrent = E_PackMLState.Idle, Message := 'Module must remain Idle during the scan that queues Start.');
		nPhase := 6;

	6:
		// Process queued Start
		LifecycleModule(
			ModuleCtrl:= ModuleCtrl,
			SystemContext:= SystemContext,
			HeartbeatIndex:= ,
			RuntimeConfig:= RuntimeConfig,
			VariableNodeReader:= VariableNodeReader,
			ServiceCtrl:= ServiceCtrl,
			ServiceParam:= ServiceParam,
			SpinAxis_BaseUnit:= SpinAxis,
			LiftPinAxis_BaseUnit:= LiftAxis);

		// Execute uses external ServiceCtrl, so Services remain Idle
		AssertTrue(Condition := LifecycleModule.PackMLOut.eStateCurrent = E_PackMLState.Execute, Message := 'Queued Start must move the Module to Execute.');
		AssertTrue(
			Condition := (LifecycleModule.ServiceStatus.SpinAxisJogCW.PackMLOut.eStateCurrent = E_PackMLState.Idle)
				AND (LifecycleModule.ServiceStatus.SpinAxisMoveAbs.PackMLOut.eStateCurrent = E_PackMLState.Idle)
				AND (LifecycleModule.ServiceStatus.SpinAxisMoveVelCW.PackMLOut.eStateCurrent = E_PackMLState.Idle)
				AND (LifecycleModule.ServiceStatus.LiftPinAxisMoveVelCW.PackMLOut.eStateCurrent = E_PackMLState.Idle)
				AND (LifecycleModule.ServiceStatus.LiftPinAxisMoveVelCCW.PackMLOut.eStateCurrent = E_PackMLState.Idle)
				AND (LifecycleModule.ServiceStatus.LiftPinAxisMoveAbs.PackMLOut.eStateCurrent = E_PackMLState.Idle),
			Message := 'Module Execute must leave Services under external control in Idle.');
		AssertTrue(Condition := (LifecycleSpinFake.CurrentCycle = 7) AND (LifecycleLiftFake.CurrentCycle = 7), Message := 'Seven Module scans must update each BaseUnit exactly seven times.');
		nPhase := 0;

		TEST_FINISHED();
END_CASE
END_METHOD

METHOD ModuleStopOverridesServiceControlAndWaitsForCleanup
VAR_INST
	SpinAxis : I_Axis_BaseUnit;
	LiftAxis : I_Axis_BaseUnit;
	HwInput : ST_Chamber1_Signal_In;
	HwOutput : ST_Chamber1_Signal_Out;
	RuntimeConfig : ST_ModuleRuntimeConfig;
	VariableNodeReader : FB_LinkVariableManager;
	ModuleCtrl : ST_ModuleCtrl;
	ServiceCtrl : ST_Chamber1_ServiceCtrl;
	ServiceParam : ST_Chamber1_ServiceParam;
	SystemContext : ST_SystemContext;
	MoveWithdrawalCall : ST_FakeAxisCall;
	StopCall : ST_FakeAxisCall;
	nHistoryBeforeStopping : UINT;
	nPhase : UINT;
END_VAR
TEST('ModuleStopOverridesServiceControlAndWaitsForCleanup');

CASE nPhase OF
	0:
		// Set Module dependencies and selected Service param
		StoppingSpinFake.M_ResetScenario();
		StoppingLiftFake.M_ResetScenario();
		SpinAxis := StoppingSpinFake;
		LiftAxis := StoppingLiftFake;
		SystemContext.UtcDateTime := '20260813123456007';
		ServiceParam.SpinAxisMoveAbs.Position := 50;
		ServiceParam.SpinAxisMoveAbs.Velocity := 10;
		ServiceParam.SpinAxisMoveAbs.Acceleration := 20;
		ServiceParam.SpinAxisMoveAbs.Deceleration := 30;

		// Initial Module scan
		StoppingModule(
			ModuleCtrl:= ModuleCtrl,
			SystemContext:= SystemContext,
			HeartbeatIndex:= ,
			RuntimeConfig:= RuntimeConfig,
			VariableNodeReader:= VariableNodeReader,
			ServiceCtrl:= ServiceCtrl,
			ServiceParam:= ServiceParam,
			SpinAxis_BaseUnit:= SpinAxis,
			LiftPinAxis_BaseUnit:= LiftAxis);
		nPhase := 1;

	1:
		// Clear Module and Services
		ModuleCtrl.PackMLIn.eCommand := E_PackMLCommand.Clear;
		ModuleCtrl.PackMLIn.bCommandChangeRequest := TRUE;
		StoppingModule(
			ModuleCtrl:= ModuleCtrl,
			SystemContext:= SystemContext,
			HeartbeatIndex:= ,
			RuntimeConfig:= RuntimeConfig,
			VariableNodeReader:= VariableNodeReader,
			ServiceCtrl:= ServiceCtrl,
			ServiceParam:= ServiceParam,
			SpinAxis_BaseUnit:= SpinAxis,
			LiftPinAxis_BaseUnit:= LiftAxis);
		nPhase := 2;

	2:
		// Finish Clearing
		ModuleCtrl.PackMLIn.bCommandChangeRequest := FALSE;
		StoppingModule(
			ModuleCtrl:= ModuleCtrl,
			SystemContext:= SystemContext,
			HeartbeatIndex:= ,
			RuntimeConfig:= RuntimeConfig,
			VariableNodeReader:= VariableNodeReader,
			ServiceCtrl:= ServiceCtrl,
			ServiceParam:= ServiceParam,
			SpinAxis_BaseUnit:= SpinAxis,
			LiftPinAxis_BaseUnit:= LiftAxis);
		nPhase := 3;

	3:
		// Reset Module and Services
		ModuleCtrl.PackMLIn.eCommand := E_PackMLCommand.Reset;
		ModuleCtrl.PackMLIn.bCommandChangeRequest := TRUE;
		StoppingModule(
			ModuleCtrl:= ModuleCtrl,
			SystemContext:= SystemContext,
			HeartbeatIndex:= ,
			RuntimeConfig:= RuntimeConfig,
			VariableNodeReader:= VariableNodeReader,
			ServiceCtrl:= ServiceCtrl,
			ServiceParam:= ServiceParam,
			SpinAxis_BaseUnit:= SpinAxis,
			LiftPinAxis_BaseUnit:= LiftAxis);
		nPhase := 4;

	4:
		// Finish Resetting
		ModuleCtrl.PackMLIn.bCommandChangeRequest := FALSE;
		StoppingModule(
			ModuleCtrl:= ModuleCtrl,
			SystemContext:= SystemContext,
			HeartbeatIndex:= ,
			RuntimeConfig:= RuntimeConfig,
			VariableNodeReader:= VariableNodeReader,
			ServiceCtrl:= ServiceCtrl,
			ServiceParam:= ServiceParam,
			SpinAxis_BaseUnit:= SpinAxis,
			LiftPinAxis_BaseUnit:= LiftAxis);
		nPhase := 5;

	5:
		// Queue Module automatic Start
		StoppingModule(
			ModuleCtrl:= ModuleCtrl,
			SystemContext:= SystemContext,
			HeartbeatIndex:= ,
			RuntimeConfig:= RuntimeConfig,
			VariableNodeReader:= VariableNodeReader,
			ServiceCtrl:= ServiceCtrl,
			ServiceParam:= ServiceParam,
			SpinAxis_BaseUnit:= SpinAxis,
			LiftPinAxis_BaseUnit:= LiftAxis);
		nPhase := 6;

	6:
		// Process Module automatic Start
		StoppingModule(
			ModuleCtrl:= ModuleCtrl,
			SystemContext:= SystemContext,
			HeartbeatIndex:= ,
			RuntimeConfig:= RuntimeConfig,
			VariableNodeReader:= VariableNodeReader,
			ServiceCtrl:= ServiceCtrl,
			ServiceParam:= ServiceParam,
			SpinAxis_BaseUnit:= SpinAxis,
			LiftPinAxis_BaseUnit:= LiftAxis);
		AssertTrue(Condition := StoppingModule.PackMLOut.eStateCurrent = E_PackMLState.Execute, Message := 'Test setup must bring the Module to Execute.');
		nPhase := 7;

	7:
		// Start SpinAxisMoveAbs through external ServiceCtrl
		ServiceCtrl.SpinAxisMoveAbs.PackMLIn.eCommand := E_PackMLCommand.Start;
		ServiceCtrl.SpinAxisMoveAbs.PackMLIn.bCommandChangeRequest := TRUE;
		StoppingModule(
			ModuleCtrl:= ModuleCtrl,
			SystemContext:= SystemContext,
			HeartbeatIndex:= ,
			RuntimeConfig:= RuntimeConfig,
			VariableNodeReader:= VariableNodeReader,
			ServiceCtrl:= ServiceCtrl,
			ServiceParam:= ServiceParam,
			SpinAxis_BaseUnit:= SpinAxis,
			LiftPinAxis_BaseUnit:= LiftAxis);
		AssertTrue(Condition := SpinAxis.M_IsResourceOwner(OwnerId := E_Chamber1ServiceId.SpinAxisMoveAbs), Message := 'Test setup must let SpinAxisMoveAbs own Spin Axis.');
		nPhase := 8;

	8:
		// Reset Service request flag and issue the active MoveAbs command
		ServiceCtrl.SpinAxisMoveAbs.PackMLIn.bCommandChangeRequest := FALSE;
		StoppingModule(
			ModuleCtrl:= ModuleCtrl,
			SystemContext:= SystemContext,
			HeartbeatIndex:= ,
			RuntimeConfig:= RuntimeConfig,
			VariableNodeReader:= VariableNodeReader,
			ServiceCtrl:= ServiceCtrl,
			ServiceParam:= ServiceParam,
			SpinAxis_BaseUnit:= SpinAxis,
			LiftPinAxis_BaseUnit:= LiftAxis);

		// Set asynchronous Stop script
		AssertTrue(
			Condition := StoppingSpinFake.M_QueueResult(
				Operation := E_FakeAxisOperation.Stop,
				AfterActiveCycles := 2,
				Done := TRUE,
				InVelocity := FALSE,
				Error := FALSE,
				ErrorId := 0),
			Message := 'Stop Done script must be accepted.');
		nPhase := 9;

	9:
		// External ServiceCtrl attempts another Start while Module requests Stop
		ServiceCtrl.SpinAxisJogCW.PackMLIn.eCommand := E_PackMLCommand.Start;
		ServiceCtrl.SpinAxisJogCW.PackMLIn.bCommandChangeRequest := TRUE;
		ModuleCtrl.RequestId := 3001;
		ModuleCtrl.PackMLIn.eCommand := E_PackMLCommand.Stop;
		ModuleCtrl.PackMLIn.bCommandChangeRequest := TRUE;
		nHistoryBeforeStopping := StoppingSpinFake.HistoryCount;

		// Cyclic update
		StoppingModule(
			ModuleCtrl:= ModuleCtrl,
			SystemContext:= SystemContext,
			HeartbeatIndex:= ,
			RuntimeConfig:= RuntimeConfig,
			VariableNodeReader:= VariableNodeReader,
			ServiceCtrl:= ServiceCtrl,
			ServiceParam:= ServiceParam,
			SpinAxis_BaseUnit:= SpinAxis,
			LiftPinAxis_BaseUnit:= LiftAxis);

